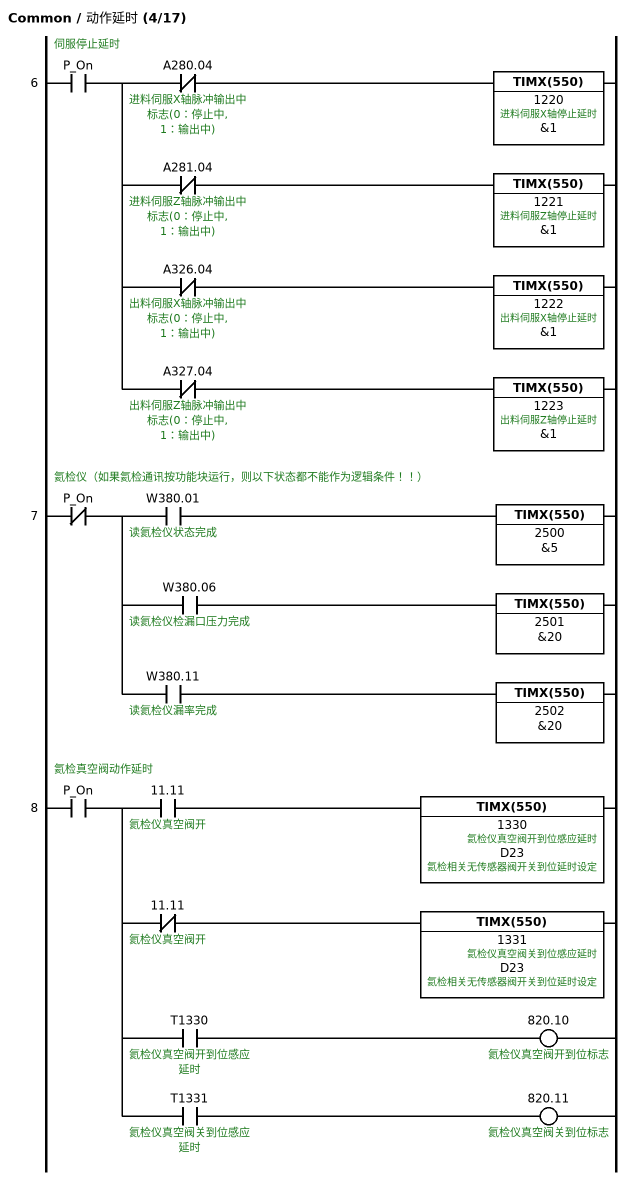
; [picture p480: Common / 动作延时, rungs 6-8]
; rung 6: 伺服停止延时
LD P_On
OUT TR0
ANDNOT A280.04  ; 进料伺服X轴脉冲输出中标志(0：停止中,1：输出中)
TIMX(550) 1220 &1  ; 进料伺服X轴停止延时
LD TR0
ANDNOT A281.04  ; 进料伺服Z轴脉冲输出中标志(0：停止中,1：输出中)
TIMX(550) 1221 &1  ; 进料伺服Z轴停止延时
LD TR0
ANDNOT A326.04  ; 出料伺服X轴脉冲输出中标志(0：停止中,1：输出中)
TIMX(550) 1222 &1  ; 出料伺服X轴停止延时
LD TR0
ANDNOT A327.04  ; 出料伺服Z轴脉冲输出中标志(0：停止中,1：输出中)
TIMX(550) 1223 &1  ; 出料伺服Z轴停止延时
; rung 7: 氦检仪（如果氦检通讯按功能块运行，则以下状态都不能作为逻辑条件！！）
LDNOT P_On
OUT TR0
AND W380.01  ; 读氦检仪状态完成
TIMX(550) 2500 &5
LD TR0
AND W380.06  ; 读氦检仪检漏口压力完成
TIMX(550) 2501 &20
LD TR0
AND W380.11  ; 读氦检仪漏率完成
TIMX(550) 2502 &20
; rung 8: 氦检真空阀动作延时
LD P_On
OUT TR0
AND 11.11  ; 氦检仪真空阀开
TIMX(550) 1330 D23  ; 氦检相关无传感器阀开关到位延时设定, 氦检仪真空阀开到位感应延时
LD TR0
ANDNOT 11.11  ; 氦检仪真空阀开
TIMX(550) 1331 D23  ; 氦检相关无传感器阀开关到位延时设定, 氦检仪真空阀关到位感应延时
LD TR0
AND T1330  ; 氦检仪真空阀开到位感应延时
OUT 820.10  ; 氦检仪真空阀开到位标志
LD TR0
AND T1331  ; 氦检仪真空阀关到位感应延时
OUT 820.11  ; 氦检仪真空阀关到位标志

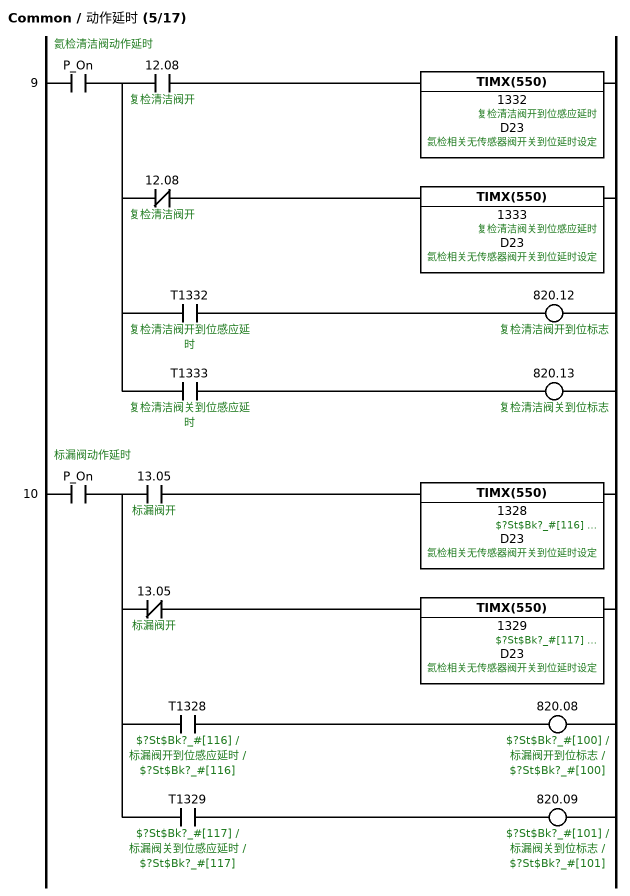
; rung 9: 氦检清洁阀动作延时
LD P_On
OUT TR0
AND 12.08  ; 复检清洁阀开
TIMX(550) 1332 D23  ; 氦检相关无传感器阀开关到位延时设定, 复检清洁阀开到位感应延时
LD TR0
ANDNOT 12.08  ; 复检清洁阀开
TIMX(550) 1333 D23  ; 氦检相关无传感器阀开关到位延时设定, 复检清洁阀关到位感应延时
LD TR0
AND T1332  ; 复检清洁阀开到位感应延时
OUT 820.12  ; 复检清洁阀开到位标志
LD TR0
AND T1333  ; 复检清洁阀关到位感应延时
OUT 820.13  ; 复检清洁阀关到位标志
; rung 10: 标漏阀动作延时
LD P_On
OUT TR0
AND 13.05  ; 标漏阀开
TIMX(550) 1328 D23  ; 氦检相关无传感器阀开关到位延时设定, $?St$Bk?_#[116] / 标漏阀开到位感应延时 / $?St$Bk?_#[116]
LD TR0
ANDNOT 13.05  ; 标漏阀开
TIMX(550) 1329 D23  ; 氦检相关无传感器阀开关到位延时设定, $?St$Bk?_#[117] / 标漏阀关到位感应延时 / $?St$Bk?_#[117]
LD TR0
AND T1328  ; $?St$Bk?_#[116] / 标漏阀开到位感应延时 / $?St$Bk?_#[116]
OUT 820.08  ; $?St$Bk?_#[100] / 标漏阀开到位标志 / $?St$Bk?_#[100]
LD TR0
AND T1329  ; $?St$Bk?_#[117] / 标漏阀关到位感应延时 / $?St$Bk?_#[117]
OUT 820.09  ; $?St$Bk?_#[101] / 标漏阀关到位标志 / $?St$Bk?_#[101]

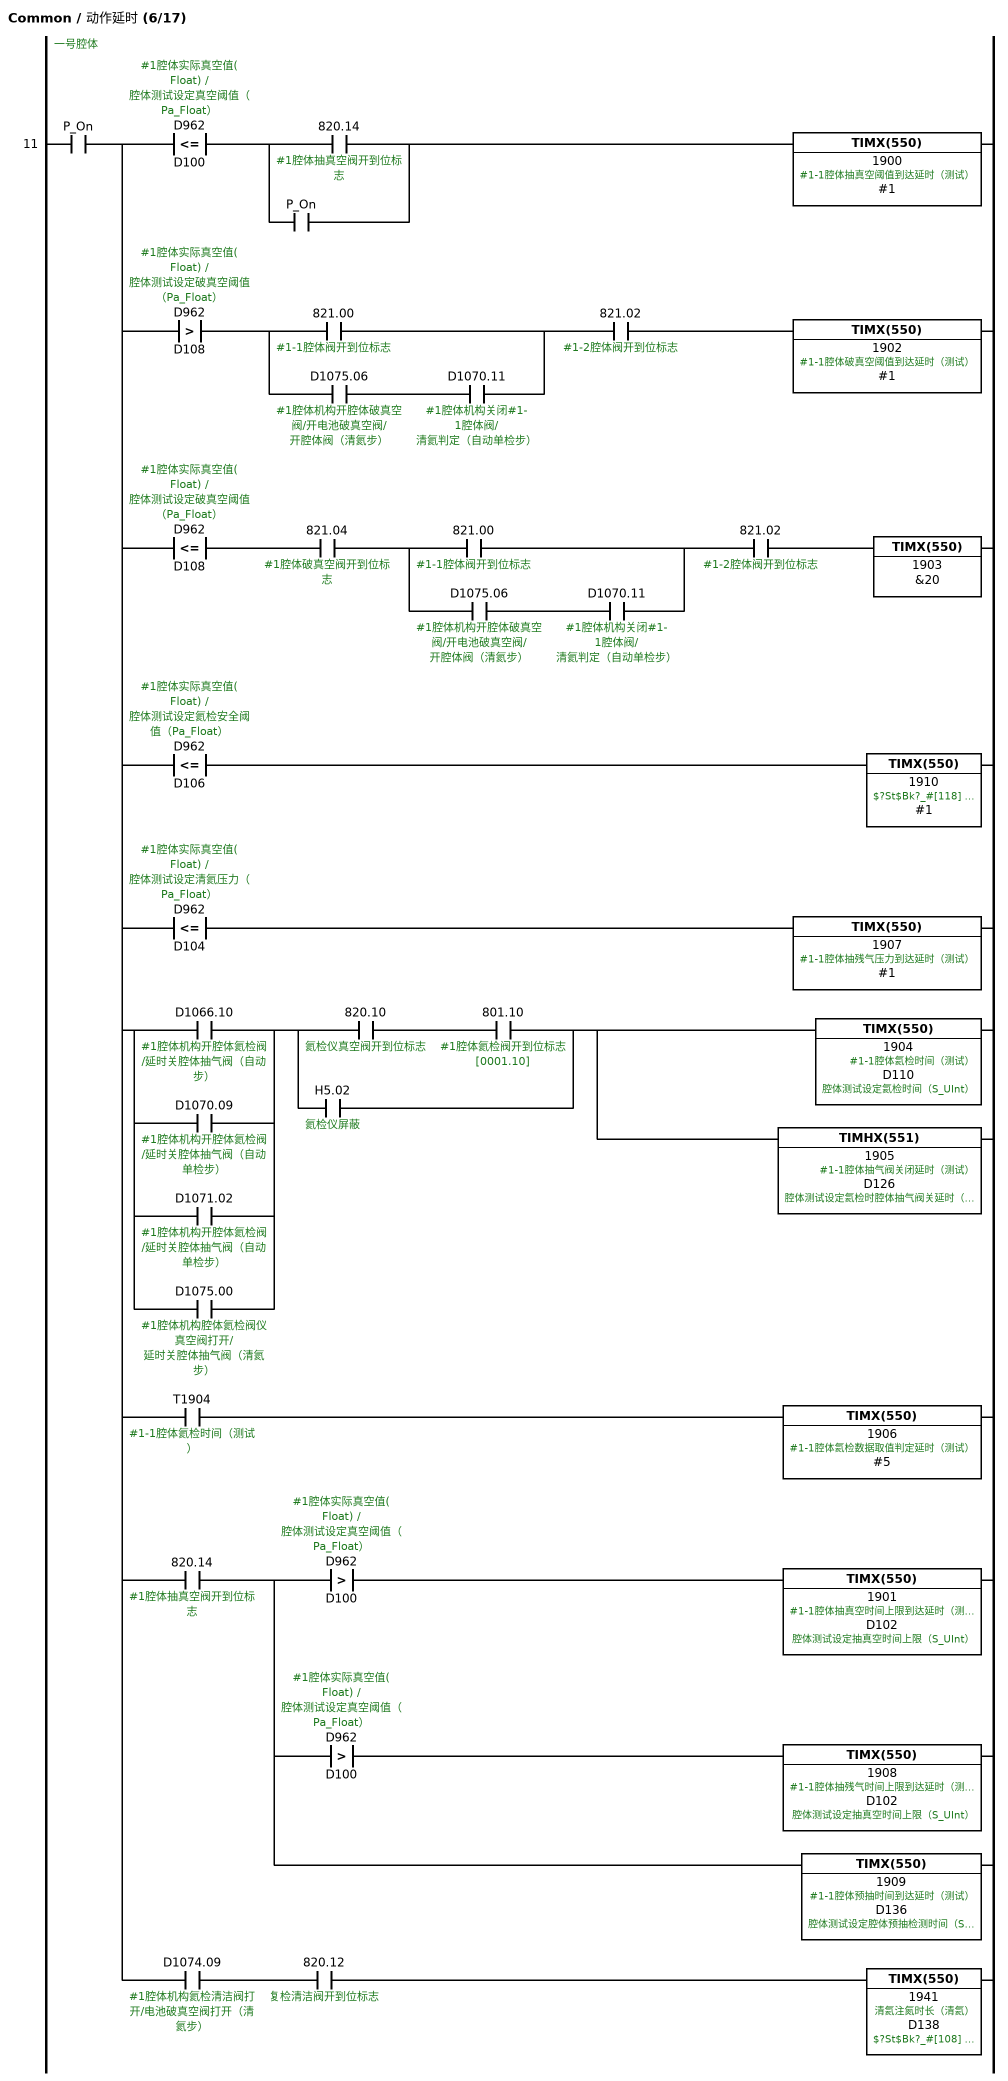
; rung 11: 一号腔体
LD P_On
OUT TR0
AND<=F(332) D962 D100  ; #1腔体实际真空值(Float), 腔体测试设定真空阈值（Pa_Float）
LD 820.14  ; #1腔体抽真空阀开到位标志
OR P_On
ANDLD
TIMX(550) 1900 #1  ; #1-1腔体抽真空阈值到达延时（测试）
LD TR0
AND>F(333) D962 D108  ; #1腔体实际真空值(Float), 腔体测试设定破真空阈值（Pa_Float）
LD 821.00  ; #1-1腔体阀开到位标志
LD D1075.06  ; #1腔体机构开腔体破真空阀/开电池破真空阀/开腔体阀（清氦步）
AND D1070.11  ; #1腔体机构关闭#1-1腔体阀/清氦判定（自动单检步）
ORLD
ANDLD
AND 821.02  ; #1-2腔体阀开到位标志
TIMX(550) 1902 #1  ; #1-1腔体破真空阈值到达延时（测试）
LD TR0
AND<=F(332) D962 D108  ; #1腔体实际真空值(Float), 腔体测试设定破真空阈值（Pa_Float）
AND 821.04  ; #1腔体破真空阀开到位标志
LD 821.00  ; #1-1腔体阀开到位标志
LD D1075.06  ; #1腔体机构开腔体破真空阀/开电池破真空阀/开腔体阀（清氦步）
AND D1070.11  ; #1腔体机构关闭#1-1腔体阀/清氦判定（自动单检步）
ORLD
ANDLD
AND 821.02  ; #1-2腔体阀开到位标志
TIMX(550) 1903 &20
LD TR0
AND<=F(332) D962 D106  ; #1腔体实际真空值(Float), 腔体测试设定氦检安全阈值（Pa_Float）
TIMX(550) 1910 #1  ; $?St$Bk?_#[118] / #1-1腔体真空在可氦检状态（测试） / $?St$Bk?_#[118]
LD TR0
AND<=F(332) D962 D104  ; #1腔体实际真空值(Float), 腔体测试设定清氦压力（Pa_Float）
TIMX(550) 1907 #1  ; #1-1腔体抽残气压力到达延时（测试）
LD TR0
LD D1066.10  ; #1腔体机构开腔体氦检阀/延时关腔体抽气阀（自动步）
OR D1070.09  ; #1腔体机构开腔体氦检阀/延时关腔体抽气阀（自动单检步）
OR D1071.02  ; #1腔体机构开腔体氦检阀/延时关腔体抽气阀（自动单检步）
OR D1075.00  ; #1腔体机构腔体氦检阀仪真空阀打开/延时关腔体抽气阀（清氦步）
ANDLD
LD 820.10  ; 氦检仪真空阀开到位标志
AND 801.10  ; #1腔体氦检阀开到位标志[0001.10]
OR H5.02  ; 氦检仪屏蔽
ANDLD
TIMX(550) 1904 D110  ; 腔体测试设定氦检时间（S_UInt）, #1-1腔体氦检时间（测试）
TIMHX(551) 1905 D126  ; 腔体测试设定氦检时腔体抽气阀关延时（S_UInt）, #1-1腔体抽气阀关闭延时（测试）
LD TR0
AND T1904  ; #1-1腔体氦检时间（测试）
TIMX(550) 1906 #5  ; #1-1腔体氦检数据取值判定延时（测试）
LD TR0
AND 820.14  ; #1腔体抽真空阀开到位标志
OUT TR1
AND>F(333) D962 D100  ; #1腔体实际真空值(Float), 腔体测试设定真空阈值（Pa_Float）
TIMX(550) 1901 D102  ; 腔体测试设定抽真空时间上限（S_UInt）, #1-1腔体抽真空时间上限到达延时（测试）
LD TR1
AND>F(333) D962 D100  ; #1腔体实际真空值(Float), 腔体测试设定真空阈值（Pa_Float）
TIMX(550) 1908 D102  ; 腔体测试设定抽真空时间上限（S_UInt）, #1-1腔体抽残气时间上限到达延时（测试）
LD TR1
TIMX(550) 1909 D136  ; 腔体测试设定腔体预抽检测时间（S_UInt）, #1-1腔体预抽时间到达延时（测试）
LD TR0
AND D1074.09  ; #1腔体机构氦检清洁阀打开/电池破真空阀打开（清氦步）
AND 820.12  ; 复检清洁阀开到位标志
TIMX(550) 1941 D138  ; $?St$Bk?_#[108] / 管路清氦注氮时间（S_UInt） / $?St$Bk?_#[108], 清氦注氮时长（清氦）

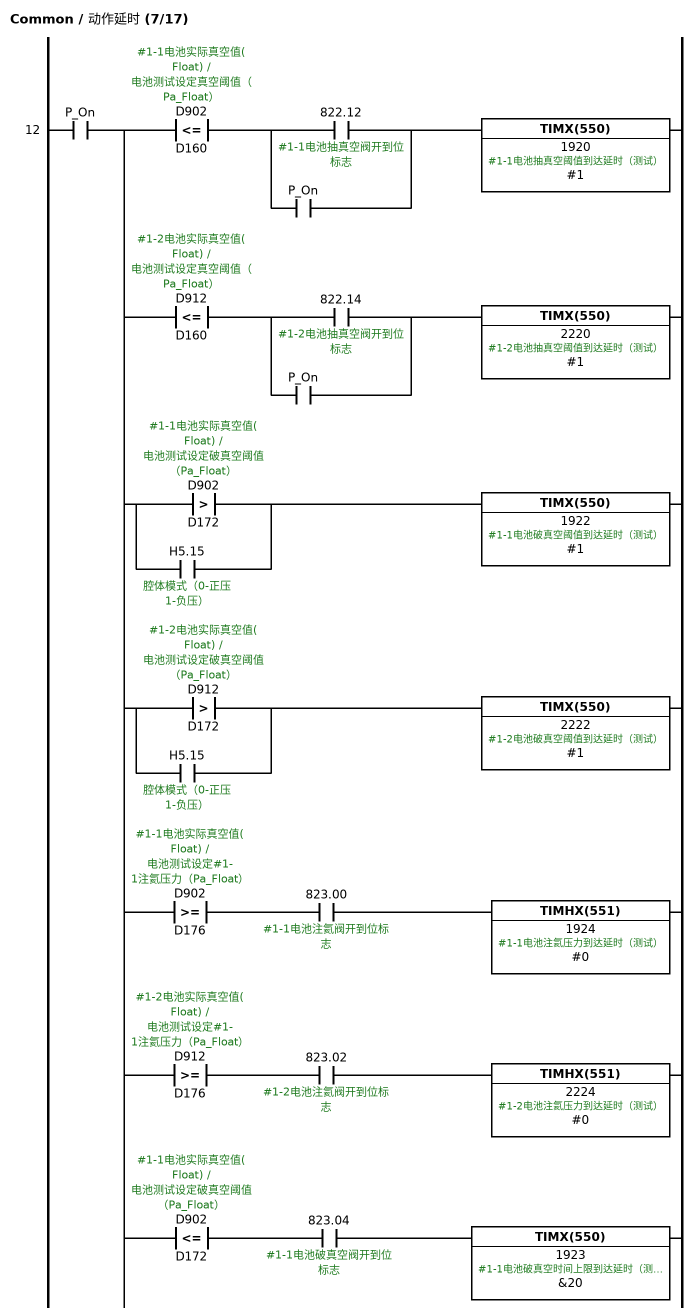

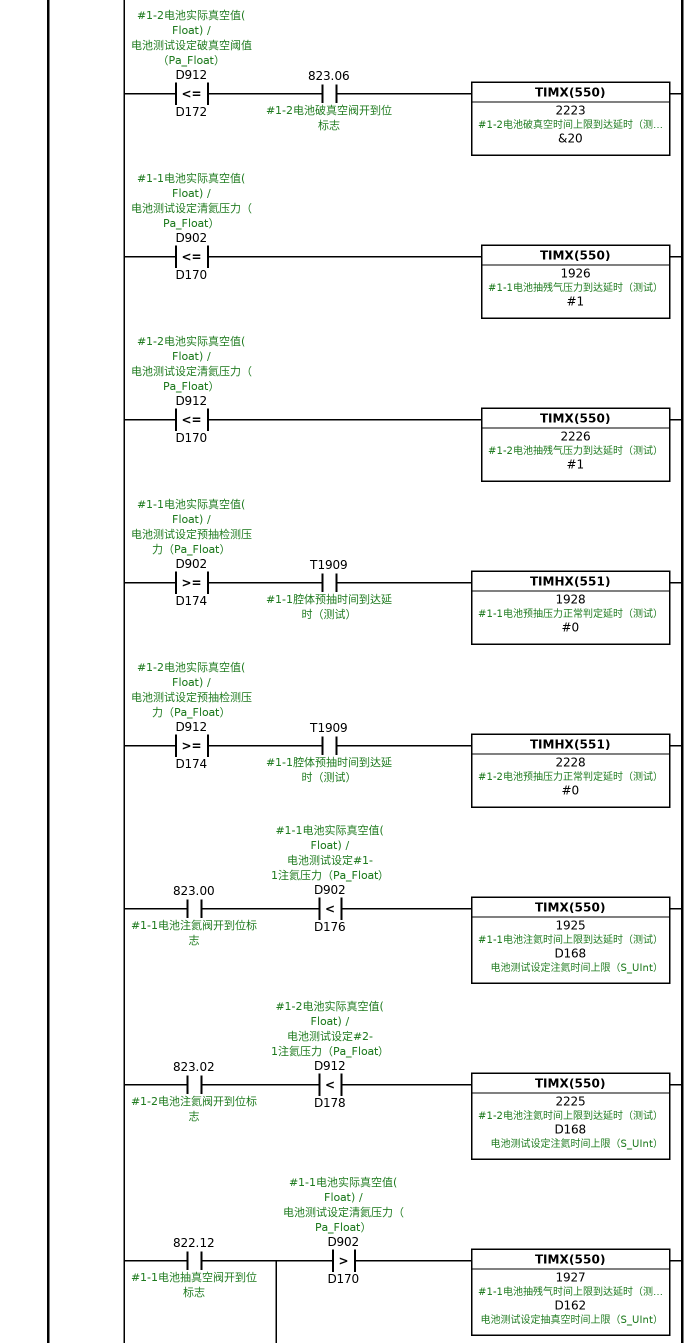

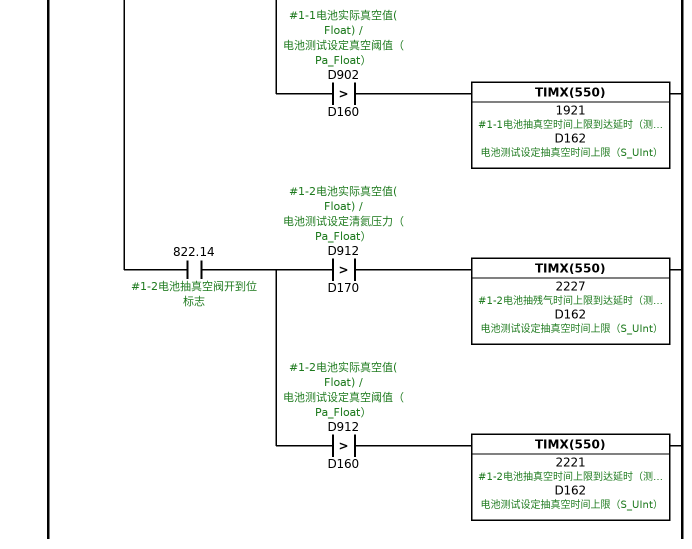
; rung 12
LD P_On
OUT TR0
AND<=F(332) D902 D160  ; #1-1电池实际真空值(Float), 电池测试设定真空阈值（Pa_Float）
LD 822.12  ; #1-1电池抽真空阀开到位标志
OR P_On
ANDLD
TIMX(550) 1920 #1  ; #1-1电池抽真空阈值到达延时（测试）
LD TR0
AND<=F(332) D912 D160  ; #1-2电池实际真空值(Float), 电池测试设定真空阈值（Pa_Float）
LD 822.14  ; #1-2电池抽真空阀开到位标志
OR P_On
ANDLD
TIMX(550) 2220 #1  ; #1-2电池抽真空阈值到达延时（测试）
LD TR0
LD>F(333) D902 D172  ; #1-1电池实际真空值(Float), 电池测试设定破真空阈值（Pa_Float）
OR H5.15  ; 腔体模式（0-正压 1-负压）
ANDLD
TIMX(550) 1922 #1  ; #1-1电池破真空阈值到达延时（测试）
LD TR0
LD>F(333) D912 D172  ; #1-2电池实际真空值(Float), 电池测试设定破真空阈值（Pa_Float）
OR H5.15  ; 腔体模式（0-正压 1-负压）
ANDLD
TIMX(550) 2222 #1  ; #1-2电池破真空阈值到达延时（测试）
LD TR0
AND>=F(334) D902 D176  ; #1-1电池实际真空值(Float), 电池测试设定#1-1注氦压力（Pa_Float）
AND 823.00  ; #1-1电池注氦阀开到位标志
TIMHX(551) 1924 #0  ; #1-1电池注氦压力到达延时（测试）
LD TR0
AND>=F(334) D912 D176  ; #1-2电池实际真空值(Float), 电池测试设定#1-1注氦压力（Pa_Float）
AND 823.02  ; #1-2电池注氦阀开到位标志
TIMHX(551) 2224 #0  ; #1-2电池注氦压力到达延时（测试）
LD TR0
AND<=F(332) D902 D172  ; #1-1电池实际真空值(Float), 电池测试设定破真空阈值（Pa_Float）
AND 823.04  ; #1-1电池破真空阀开到位标志
TIMX(550) 1923 &20  ; #1-1电池破真空时间上限到达延时（测试）
LD TR0
AND<=F(332) D912 D172  ; #1-2电池实际真空值(Float), 电池测试设定破真空阈值（Pa_Float）
AND 823.06  ; #1-2电池破真空阀开到位标志
TIMX(550) 2223 &20  ; #1-2电池破真空时间上限到达延时（测试）
LD TR0
AND<=F(332) D902 D170  ; #1-1电池实际真空值(Float), 电池测试设定清氦压力（Pa_Float）
TIMX(550) 1926 #1  ; #1-1电池抽残气压力到达延时（测试）
LD TR0
AND<=F(332) D912 D170  ; #1-2电池实际真空值(Float), 电池测试设定清氦压力（Pa_Float）
TIMX(550) 2226 #1  ; #1-2电池抽残气压力到达延时（测试）
LD TR0
AND>=F(334) D902 D174  ; #1-1电池实际真空值(Float), 电池测试设定预抽检测压力（Pa_Float）
AND T1909  ; #1-1腔体预抽时间到达延时（测试）
TIMHX(551) 1928 #0  ; #1-1电池预抽压力正常判定延时（测试）
LD TR0
AND>=F(334) D912 D174  ; #1-2电池实际真空值(Float), 电池测试设定预抽检测压力（Pa_Float）
AND T1909  ; #1-1腔体预抽时间到达延时（测试）
TIMHX(551) 2228 #0  ; #1-2电池预抽压力正常判定延时（测试）
LD TR0
AND 823.00  ; #1-1电池注氦阀开到位标志
AND<F(331) D902 D176  ; #1-1电池实际真空值(Float), 电池测试设定#1-1注氦压力（Pa_Float）
TIMX(550) 1925 D168  ; 电池测试设定注氦时间上限（S_UInt）, #1-1电池注氦时间上限到达延时（测试）
LD TR0
AND 823.02  ; #1-2电池注氦阀开到位标志
AND<F(331) D912 D178  ; #1-2电池实际真空值(Float), 电池测试设定#2-1注氦压力（Pa_Float）
TIMX(550) 2225 D168  ; 电池测试设定注氦时间上限（S_UInt）, #1-2电池注氦时间上限到达延时（测试）
LD TR0
AND 822.12  ; #1-1电池抽真空阀开到位标志
OUT TR1
AND>F(333) D902 D170  ; #1-1电池实际真空值(Float), 电池测试设定清氦压力（Pa_Float）
TIMX(550) 1927 D162  ; 电池测试设定抽真空时间上限（S_UInt）, #1-1电池抽残气时间上限到达延时（测试）
LD TR1
AND>F(333) D902 D160  ; #1-1电池实际真空值(Float), 电池测试设定真空阈值（Pa_Float）
TIMX(550) 1921 D162  ; 电池测试设定抽真空时间上限（S_UInt）, #1-1电池抽真空时间上限到达延时（测试）
LD TR0
AND 822.14  ; #1-2电池抽真空阀开到位标志
OUT TR0
AND>F(333) D912 D170  ; #1-2电池实际真空值(Float), 电池测试设定清氦压力（Pa_Float）
TIMX(550) 2227 D162  ; 电池测试设定抽真空时间上限（S_UInt）, #1-2电池抽残气时间上限到达延时（测试）
LD TR0
AND>F(333) D912 D160  ; #1-2电池实际真空值(Float), 电池测试设定真空阈值（Pa_Float）
TIMX(550) 2221 D162  ; 电池测试设定抽真空时间上限（S_UInt）, #1-2电池抽真空时间上限到达延时（测试）

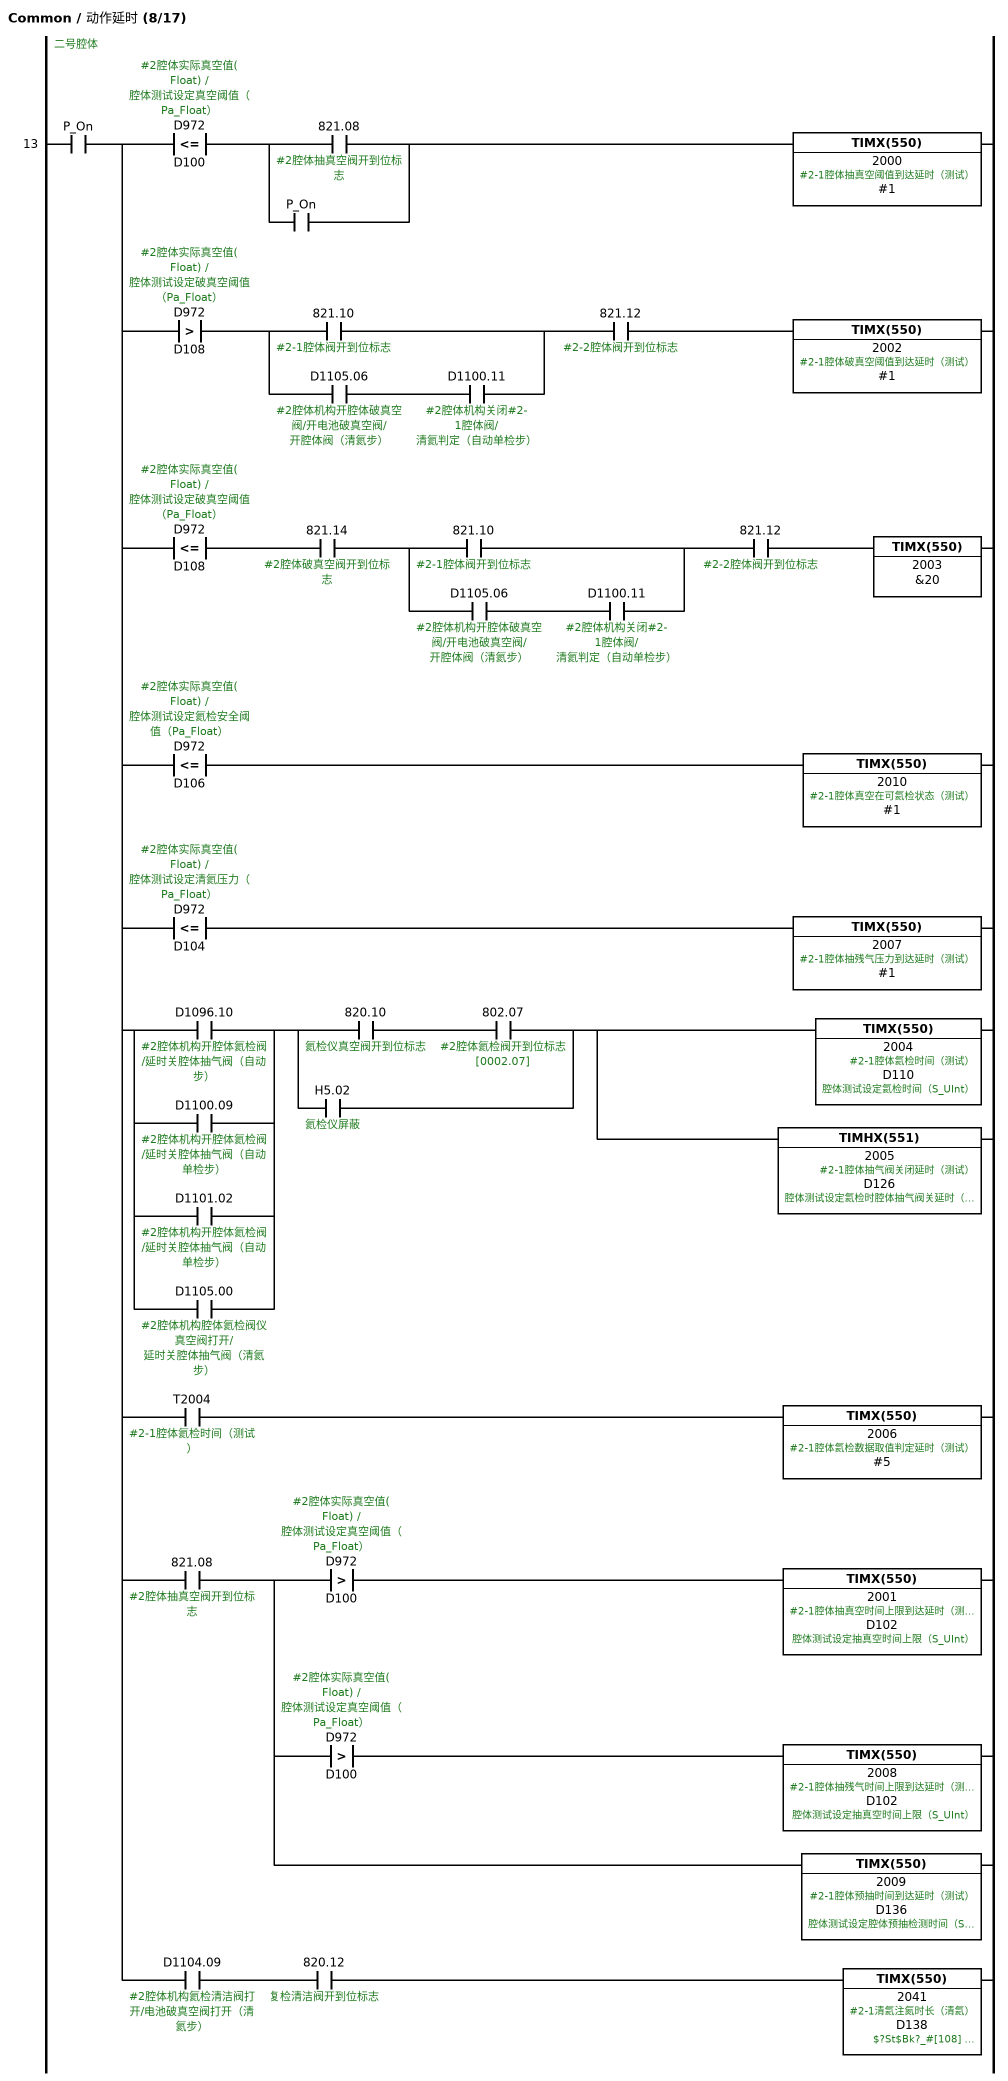
; rung 13: 二号腔体
LD P_On
OUT TR0
AND<=F(332) D972 D100  ; #2腔体实际真空值(Float), 腔体测试设定真空阈值（Pa_Float）
LD 821.08  ; #2腔体抽真空阀开到位标志
OR P_On
ANDLD
TIMX(550) 2000 #1  ; #2-1腔体抽真空阈值到达延时（测试）
LD TR0
AND>F(333) D972 D108  ; #2腔体实际真空值(Float), 腔体测试设定破真空阈值（Pa_Float）
LD 821.10  ; #2-1腔体阀开到位标志
LD D1105.06  ; #2腔体机构开腔体破真空阀/开电池破真空阀/开腔体阀（清氦步）
AND D1100.11  ; #2腔体机构关闭#2-1腔体阀/清氦判定（自动单检步）
ORLD
ANDLD
AND 821.12  ; #2-2腔体阀开到位标志
TIMX(550) 2002 #1  ; #2-1腔体破真空阈值到达延时（测试）
LD TR0
AND<=F(332) D972 D108  ; #2腔体实际真空值(Float), 腔体测试设定破真空阈值（Pa_Float）
AND 821.14  ; #2腔体破真空阀开到位标志
LD 821.10  ; #2-1腔体阀开到位标志
LD D1105.06  ; #2腔体机构开腔体破真空阀/开电池破真空阀/开腔体阀（清氦步）
AND D1100.11  ; #2腔体机构关闭#2-1腔体阀/清氦判定（自动单检步）
ORLD
ANDLD
AND 821.12  ; #2-2腔体阀开到位标志
TIMX(550) 2003 &20
LD TR0
AND<=F(332) D972 D106  ; #2腔体实际真空值(Float), 腔体测试设定氦检安全阈值（Pa_Float）
TIMX(550) 2010 #1  ; #2-1腔体真空在可氦检状态（测试）
LD TR0
AND<=F(332) D972 D104  ; #2腔体实际真空值(Float), 腔体测试设定清氦压力（Pa_Float）
TIMX(550) 2007 #1  ; #2-1腔体抽残气压力到达延时（测试）
LD TR0
LD D1096.10  ; #2腔体机构开腔体氦检阀/延时关腔体抽气阀（自动步）
OR D1100.09  ; #2腔体机构开腔体氦检阀/延时关腔体抽气阀（自动单检步）
OR D1101.02  ; #2腔体机构开腔体氦检阀/延时关腔体抽气阀（自动单检步）
OR D1105.00  ; #2腔体机构腔体氦检阀仪真空阀打开/延时关腔体抽气阀（清氦步）
ANDLD
LD 820.10  ; 氦检仪真空阀开到位标志
AND 802.07  ; #2腔体氦检阀开到位标志[0002.07]
OR H5.02  ; 氦检仪屏蔽
ANDLD
TIMX(550) 2004 D110  ; 腔体测试设定氦检时间（S_UInt）, #2-1腔体氦检时间（测试）
TIMHX(551) 2005 D126  ; 腔体测试设定氦检时腔体抽气阀关延时（S_UInt）, #2-1腔体抽气阀关闭延时（测试）
LD TR0
AND T2004  ; #2-1腔体氦检时间（测试）
TIMX(550) 2006 #5  ; #2-1腔体氦检数据取值判定延时（测试）
LD TR0
AND 821.08  ; #2腔体抽真空阀开到位标志
OUT TR1
AND>F(333) D972 D100  ; #2腔体实际真空值(Float), 腔体测试设定真空阈值（Pa_Float）
TIMX(550) 2001 D102  ; 腔体测试设定抽真空时间上限（S_UInt）, #2-1腔体抽真空时间上限到达延时（测试）
LD TR1
AND>F(333) D972 D100  ; #2腔体实际真空值(Float), 腔体测试设定真空阈值（Pa_Float）
TIMX(550) 2008 D102  ; 腔体测试设定抽真空时间上限（S_UInt）, #2-1腔体抽残气时间上限到达延时（测试）
LD TR1
TIMX(550) 2009 D136  ; 腔体测试设定腔体预抽检测时间（S_UInt）, #2-1腔体预抽时间到达延时（测试）
LD TR0
AND D1104.09  ; #2腔体机构氦检清洁阀打开/电池破真空阀打开（清氦步）
AND 820.12  ; 复检清洁阀开到位标志
TIMX(550) 2041 D138  ; $?St$Bk?_#[108] / 管路清氦注氮时间（S_UInt） / $?St$Bk?_#[108], #2-1清氦注氮时长（清氦）

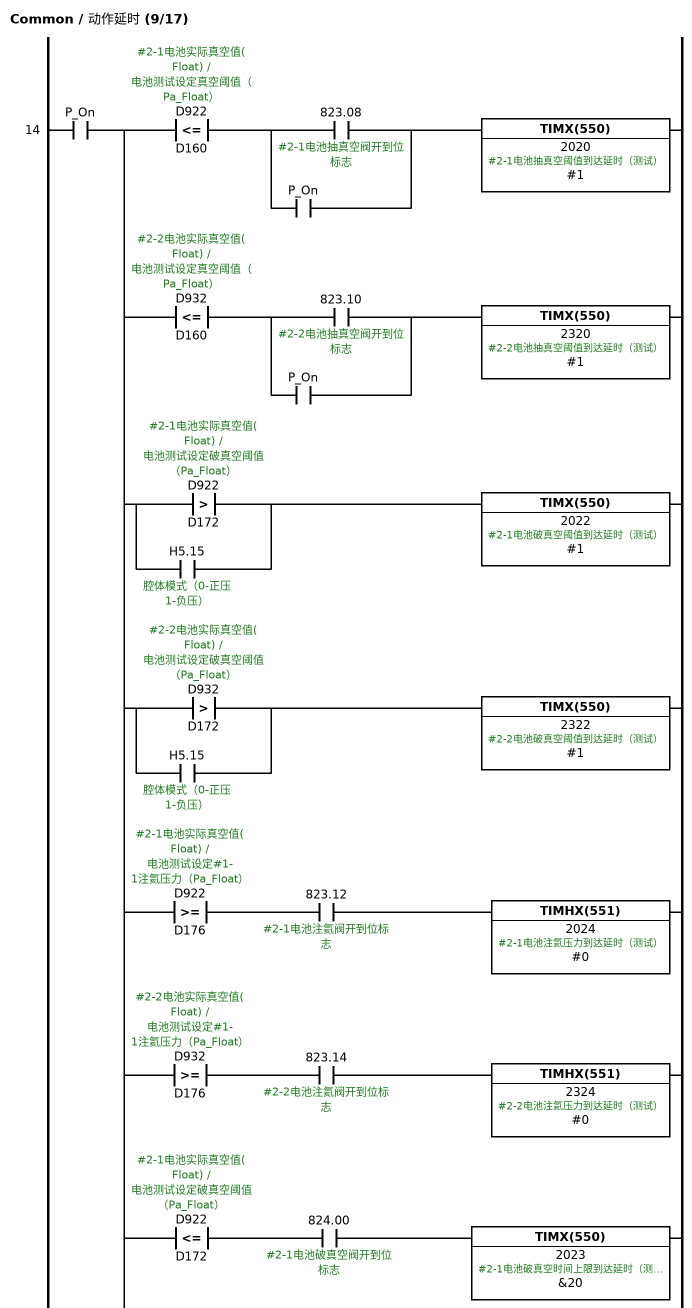

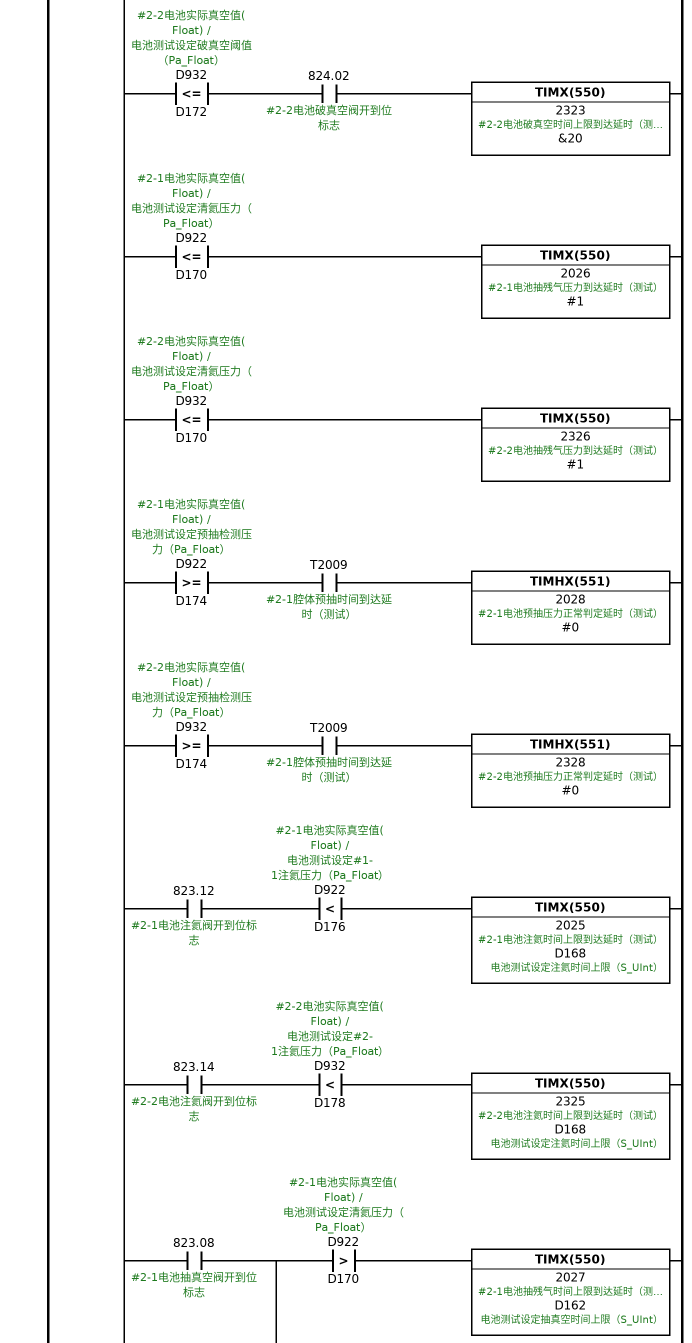

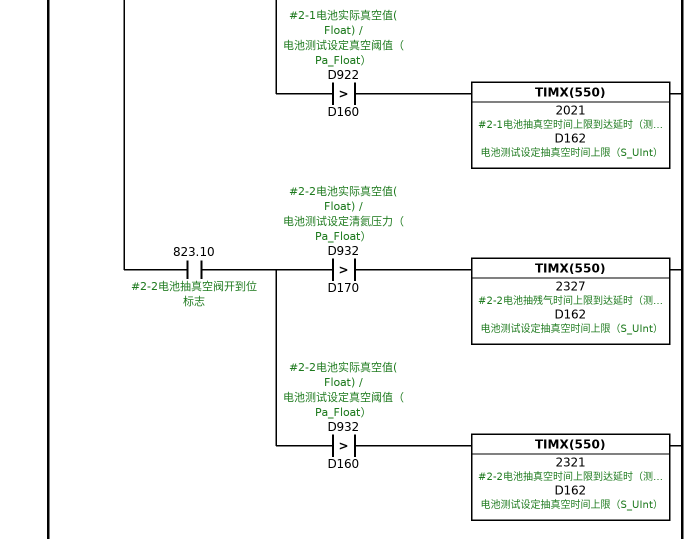
; rung 14
LD P_On
OUT TR0
AND<=F(332) D922 D160  ; #2-1电池实际真空值(Float), 电池测试设定真空阈值（Pa_Float）
LD 823.08  ; #2-1电池抽真空阀开到位标志
OR P_On
ANDLD
TIMX(550) 2020 #1  ; #2-1电池抽真空阈值到达延时（测试）
LD TR0
AND<=F(332) D932 D160  ; #2-2电池实际真空值(Float), 电池测试设定真空阈值（Pa_Float）
LD 823.10  ; #2-2电池抽真空阀开到位标志
OR P_On
ANDLD
TIMX(550) 2320 #1  ; #2-2电池抽真空阈值到达延时（测试）
LD TR0
LD>F(333) D922 D172  ; #2-1电池实际真空值(Float), 电池测试设定破真空阈值（Pa_Float）
OR H5.15  ; 腔体模式（0-正压 1-负压）
ANDLD
TIMX(550) 2022 #1  ; #2-1电池破真空阈值到达延时（测试）
LD TR0
LD>F(333) D932 D172  ; #2-2电池实际真空值(Float), 电池测试设定破真空阈值（Pa_Float）
OR H5.15  ; 腔体模式（0-正压 1-负压）
ANDLD
TIMX(550) 2322 #1  ; #2-2电池破真空阈值到达延时（测试）
LD TR0
AND>=F(334) D922 D176  ; #2-1电池实际真空值(Float), 电池测试设定#1-1注氦压力（Pa_Float）
AND 823.12  ; #2-1电池注氦阀开到位标志
TIMHX(551) 2024 #0  ; #2-1电池注氦压力到达延时（测试）
LD TR0
AND>=F(334) D932 D176  ; #2-2电池实际真空值(Float), 电池测试设定#1-1注氦压力（Pa_Float）
AND 823.14  ; #2-2电池注氦阀开到位标志
TIMHX(551) 2324 #0  ; #2-2电池注氦压力到达延时（测试）
LD TR0
AND<=F(332) D922 D172  ; #2-1电池实际真空值(Float), 电池测试设定破真空阈值（Pa_Float）
AND 824.00  ; #2-1电池破真空阀开到位标志
TIMX(550) 2023 &20  ; #2-1电池破真空时间上限到达延时（测试）
LD TR0
AND<=F(332) D932 D172  ; #2-2电池实际真空值(Float), 电池测试设定破真空阈值（Pa_Float）
AND 824.02  ; #2-2电池破真空阀开到位标志
TIMX(550) 2323 &20  ; #2-2电池破真空时间上限到达延时（测试）
LD TR0
AND<=F(332) D922 D170  ; #2-1电池实际真空值(Float), 电池测试设定清氦压力（Pa_Float）
TIMX(550) 2026 #1  ; #2-1电池抽残气压力到达延时（测试）
LD TR0
AND<=F(332) D932 D170  ; #2-2电池实际真空值(Float), 电池测试设定清氦压力（Pa_Float）
TIMX(550) 2326 #1  ; #2-2电池抽残气压力到达延时（测试）
LD TR0
AND>=F(334) D922 D174  ; #2-1电池实际真空值(Float), 电池测试设定预抽检测压力（Pa_Float）
AND T2009  ; #2-1腔体预抽时间到达延时（测试）
TIMHX(551) 2028 #0  ; #2-1电池预抽压力正常判定延时（测试）
LD TR0
AND>=F(334) D932 D174  ; #2-2电池实际真空值(Float), 电池测试设定预抽检测压力（Pa_Float）
AND T2009  ; #2-1腔体预抽时间到达延时（测试）
TIMHX(551) 2328 #0  ; #2-2电池预抽压力正常判定延时（测试）
LD TR0
AND 823.12  ; #2-1电池注氦阀开到位标志
AND<F(331) D922 D176  ; #2-1电池实际真空值(Float), 电池测试设定#1-1注氦压力（Pa_Float）
TIMX(550) 2025 D168  ; 电池测试设定注氦时间上限（S_UInt）, #2-1电池注氦时间上限到达延时（测试）
LD TR0
AND 823.14  ; #2-2电池注氦阀开到位标志
AND<F(331) D932 D178  ; #2-2电池实际真空值(Float), 电池测试设定#2-1注氦压力（Pa_Float）
TIMX(550) 2325 D168  ; 电池测试设定注氦时间上限（S_UInt）, #2-2电池注氦时间上限到达延时（测试）
LD TR0
AND 823.08  ; #2-1电池抽真空阀开到位标志
OUT TR1
AND>F(333) D922 D170  ; #2-1电池实际真空值(Float), 电池测试设定清氦压力（Pa_Float）
TIMX(550) 2027 D162  ; 电池测试设定抽真空时间上限（S_UInt）, #2-1电池抽残气时间上限到达延时（测试）
LD TR1
AND>F(333) D922 D160  ; #2-1电池实际真空值(Float), 电池测试设定真空阈值（Pa_Float）
TIMX(550) 2021 D162  ; 电池测试设定抽真空时间上限（S_UInt）, #2-1电池抽真空时间上限到达延时（测试）
LD TR0
AND 823.10  ; #2-2电池抽真空阀开到位标志
OUT TR0
AND>F(333) D932 D170  ; #2-2电池实际真空值(Float), 电池测试设定清氦压力（Pa_Float）
TIMX(550) 2327 D162  ; 电池测试设定抽真空时间上限（S_UInt）, #2-2电池抽残气时间上限到达延时（测试）
LD TR0
AND>F(333) D932 D160  ; #2-2电池实际真空值(Float), 电池测试设定真空阈值（Pa_Float）
TIMX(550) 2321 D162  ; 电池测试设定抽真空时间上限（S_UInt）, #2-2电池抽真空时间上限到达延时（测试）

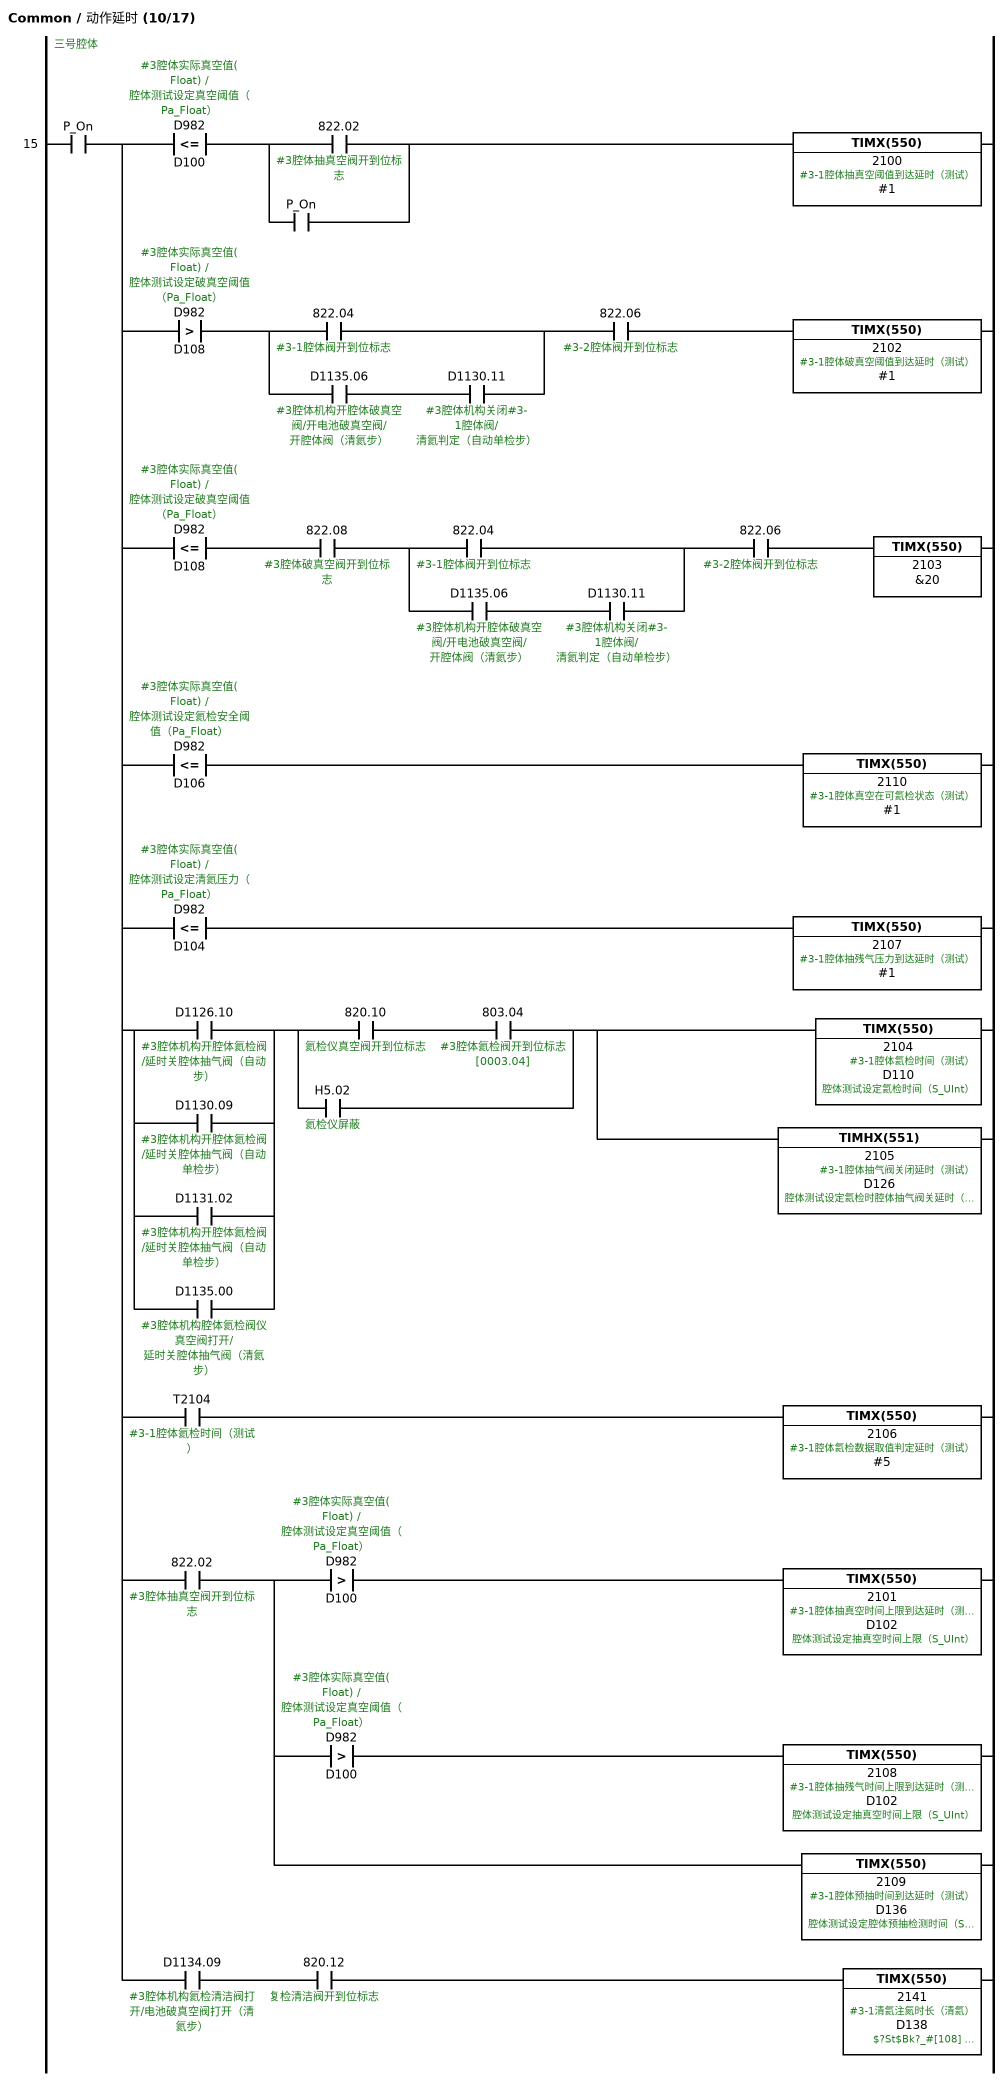
; rung 15: 三号腔体
LD P_On
OUT TR0
AND<=F(332) D982 D100  ; #3腔体实际真空值(Float), 腔体测试设定真空阈值（Pa_Float）
LD 822.02  ; #3腔体抽真空阀开到位标志
OR P_On
ANDLD
TIMX(550) 2100 #1  ; #3-1腔体抽真空阈值到达延时（测试）
LD TR0
AND>F(333) D982 D108  ; #3腔体实际真空值(Float), 腔体测试设定破真空阈值（Pa_Float）
LD 822.04  ; #3-1腔体阀开到位标志
LD D1135.06  ; #3腔体机构开腔体破真空阀/开电池破真空阀/开腔体阀（清氦步）
AND D1130.11  ; #3腔体机构关闭#3-1腔体阀/清氦判定（自动单检步）
ORLD
ANDLD
AND 822.06  ; #3-2腔体阀开到位标志
TIMX(550) 2102 #1  ; #3-1腔体破真空阈值到达延时（测试）
LD TR0
AND<=F(332) D982 D108  ; #3腔体实际真空值(Float), 腔体测试设定破真空阈值（Pa_Float）
AND 822.08  ; #3腔体破真空阀开到位标志
LD 822.04  ; #3-1腔体阀开到位标志
LD D1135.06  ; #3腔体机构开腔体破真空阀/开电池破真空阀/开腔体阀（清氦步）
AND D1130.11  ; #3腔体机构关闭#3-1腔体阀/清氦判定（自动单检步）
ORLD
ANDLD
AND 822.06  ; #3-2腔体阀开到位标志
TIMX(550) 2103 &20
LD TR0
AND<=F(332) D982 D106  ; #3腔体实际真空值(Float), 腔体测试设定氦检安全阈值（Pa_Float）
TIMX(550) 2110 #1  ; #3-1腔体真空在可氦检状态（测试）
LD TR0
AND<=F(332) D982 D104  ; #3腔体实际真空值(Float), 腔体测试设定清氦压力（Pa_Float）
TIMX(550) 2107 #1  ; #3-1腔体抽残气压力到达延时（测试）
LD TR0
LD D1126.10  ; #3腔体机构开腔体氦检阀/延时关腔体抽气阀（自动步）
OR D1130.09  ; #3腔体机构开腔体氦检阀/延时关腔体抽气阀（自动单检步）
OR D1131.02  ; #3腔体机构开腔体氦检阀/延时关腔体抽气阀（自动单检步）
OR D1135.00  ; #3腔体机构腔体氦检阀仪真空阀打开/延时关腔体抽气阀（清氦步）
ANDLD
LD 820.10  ; 氦检仪真空阀开到位标志
AND 803.04  ; #3腔体氦检阀开到位标志[0003.04]
OR H5.02  ; 氦检仪屏蔽
ANDLD
TIMX(550) 2104 D110  ; 腔体测试设定氦检时间（S_UInt）, #3-1腔体氦检时间（测试）
TIMHX(551) 2105 D126  ; 腔体测试设定氦检时腔体抽气阀关延时（S_UInt）, #3-1腔体抽气阀关闭延时（测试）
LD TR0
AND T2104  ; #3-1腔体氦检时间（测试）
TIMX(550) 2106 #5  ; #3-1腔体氦检数据取值判定延时（测试）
LD TR0
AND 822.02  ; #3腔体抽真空阀开到位标志
OUT TR1
AND>F(333) D982 D100  ; #3腔体实际真空值(Float), 腔体测试设定真空阈值（Pa_Float）
TIMX(550) 2101 D102  ; 腔体测试设定抽真空时间上限（S_UInt）, #3-1腔体抽真空时间上限到达延时（测试）
LD TR1
AND>F(333) D982 D100  ; #3腔体实际真空值(Float), 腔体测试设定真空阈值（Pa_Float）
TIMX(550) 2108 D102  ; 腔体测试设定抽真空时间上限（S_UInt）, #3-1腔体抽残气时间上限到达延时（测试）
LD TR1
TIMX(550) 2109 D136  ; 腔体测试设定腔体预抽检测时间（S_UInt）, #3-1腔体预抽时间到达延时（测试）
LD TR0
AND D1134.09  ; #3腔体机构氦检清洁阀打开/电池破真空阀打开（清氦步）
AND 820.12  ; 复检清洁阀开到位标志
TIMX(550) 2141 D138  ; $?St$Bk?_#[108] / 管路清氦注氮时间（S_UInt） / $?St$Bk?_#[108], #3-1清氦注氮时长（清氦）

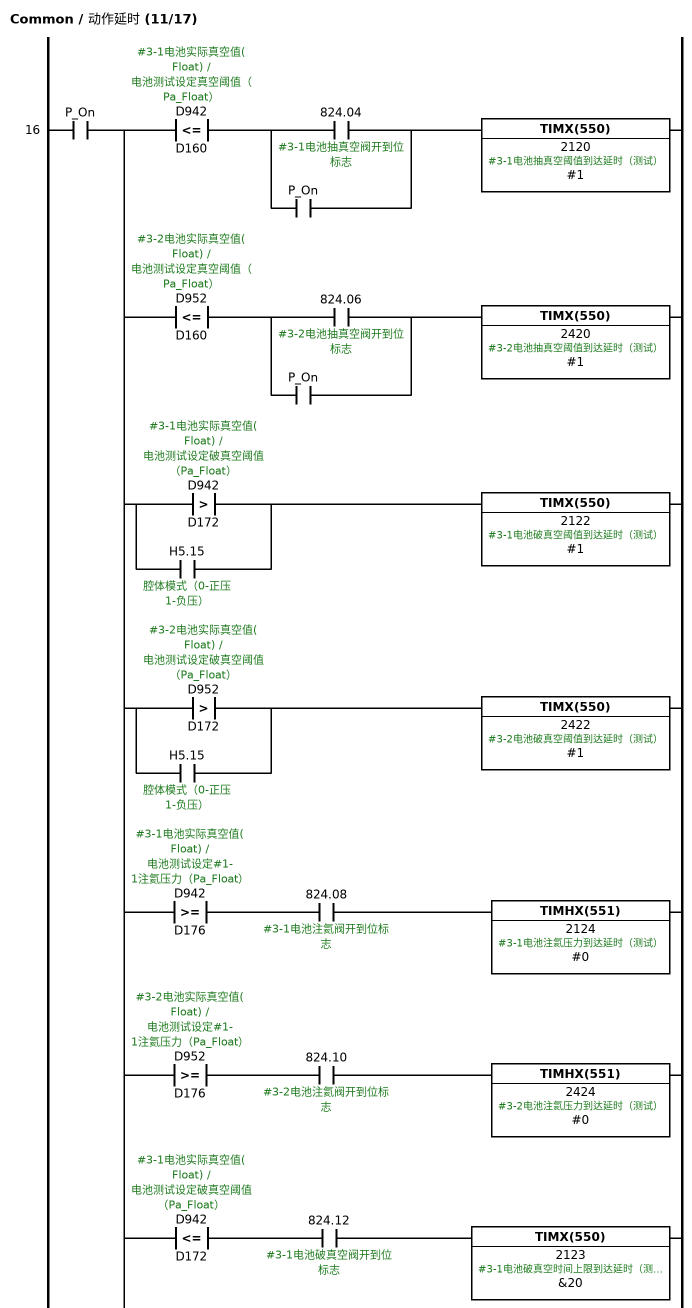

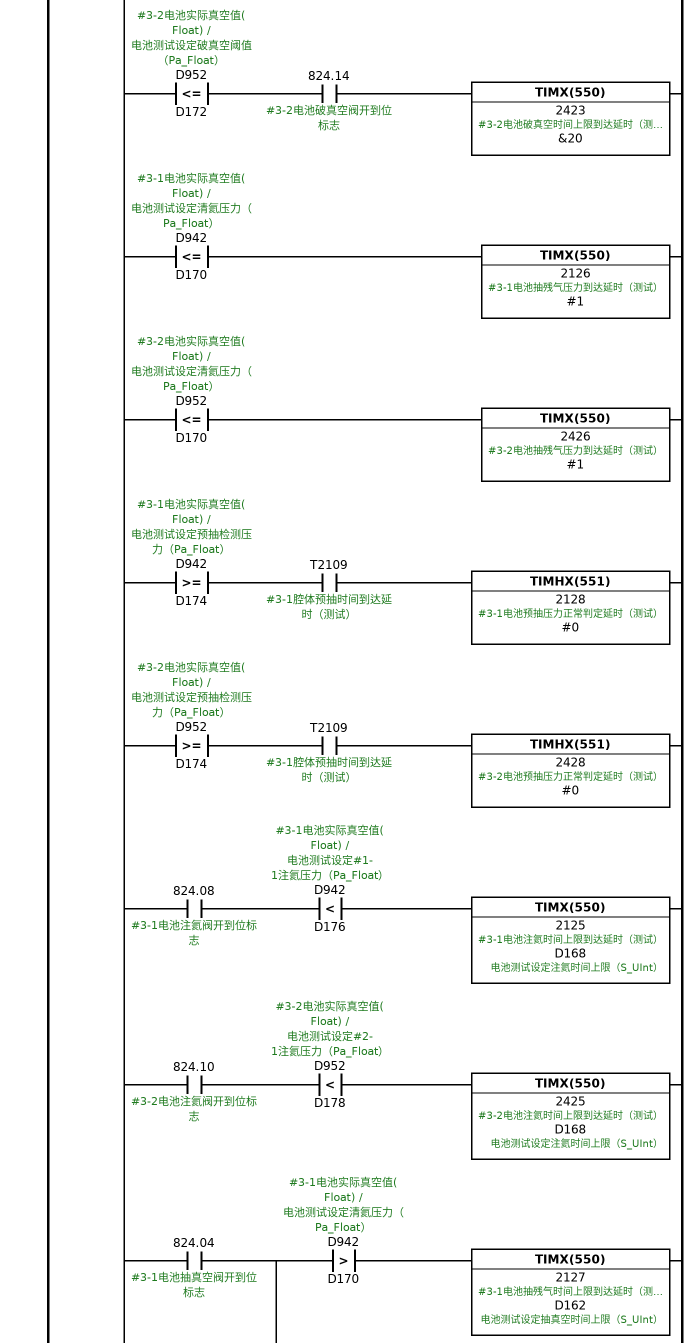

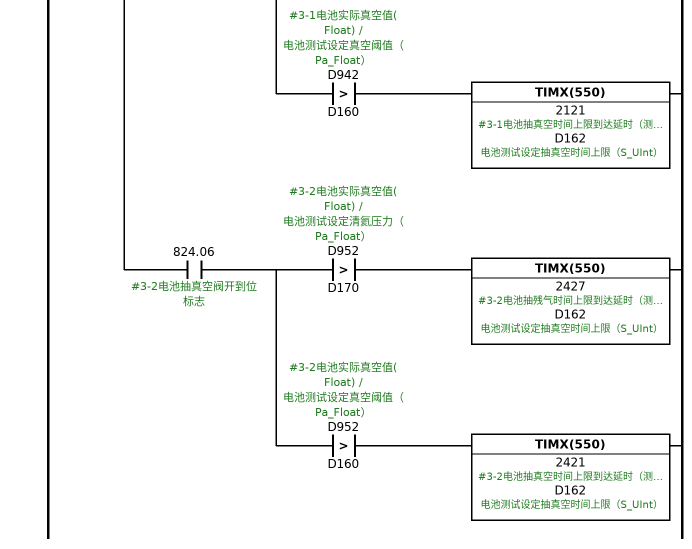
; rung 16
LD P_On
OUT TR0
AND<=F(332) D942 D160  ; #3-1电池实际真空值(Float), 电池测试设定真空阈值（Pa_Float）
LD 824.04  ; #3-1电池抽真空阀开到位标志
OR P_On
ANDLD
TIMX(550) 2120 #1  ; #3-1电池抽真空阈值到达延时（测试）
LD TR0
AND<=F(332) D952 D160  ; #3-2电池实际真空值(Float), 电池测试设定真空阈值（Pa_Float）
LD 824.06  ; #3-2电池抽真空阀开到位标志
OR P_On
ANDLD
TIMX(550) 2420 #1  ; #3-2电池抽真空阈值到达延时（测试）
LD TR0
LD>F(333) D942 D172  ; #3-1电池实际真空值(Float), 电池测试设定破真空阈值（Pa_Float）
OR H5.15  ; 腔体模式（0-正压 1-负压）
ANDLD
TIMX(550) 2122 #1  ; #3-1电池破真空阈值到达延时（测试）
LD TR0
LD>F(333) D952 D172  ; #3-2电池实际真空值(Float), 电池测试设定破真空阈值（Pa_Float）
OR H5.15  ; 腔体模式（0-正压 1-负压）
ANDLD
TIMX(550) 2422 #1  ; #3-2电池破真空阈值到达延时（测试）
LD TR0
AND>=F(334) D942 D176  ; #3-1电池实际真空值(Float), 电池测试设定#1-1注氦压力（Pa_Float）
AND 824.08  ; #3-1电池注氦阀开到位标志
TIMHX(551) 2124 #0  ; #3-1电池注氦压力到达延时（测试）
LD TR0
AND>=F(334) D952 D176  ; #3-2电池实际真空值(Float), 电池测试设定#1-1注氦压力（Pa_Float）
AND 824.10  ; #3-2电池注氦阀开到位标志
TIMHX(551) 2424 #0  ; #3-2电池注氦压力到达延时（测试）
LD TR0
AND<=F(332) D942 D172  ; #3-1电池实际真空值(Float), 电池测试设定破真空阈值（Pa_Float）
AND 824.12  ; #3-1电池破真空阀开到位标志
TIMX(550) 2123 &20  ; #3-1电池破真空时间上限到达延时（测试）
LD TR0
AND<=F(332) D952 D172  ; #3-2电池实际真空值(Float), 电池测试设定破真空阈值（Pa_Float）
AND 824.14  ; #3-2电池破真空阀开到位标志
TIMX(550) 2423 &20  ; #3-2电池破真空时间上限到达延时（测试）
LD TR0
AND<=F(332) D942 D170  ; #3-1电池实际真空值(Float), 电池测试设定清氦压力（Pa_Float）
TIMX(550) 2126 #1  ; #3-1电池抽残气压力到达延时（测试）
LD TR0
AND<=F(332) D952 D170  ; #3-2电池实际真空值(Float), 电池测试设定清氦压力（Pa_Float）
TIMX(550) 2426 #1  ; #3-2电池抽残气压力到达延时（测试）
LD TR0
AND>=F(334) D942 D174  ; #3-1电池实际真空值(Float), 电池测试设定预抽检测压力（Pa_Float）
AND T2109  ; #3-1腔体预抽时间到达延时（测试）
TIMHX(551) 2128 #0  ; #3-1电池预抽压力正常判定延时（测试）
LD TR0
AND>=F(334) D952 D174  ; #3-2电池实际真空值(Float), 电池测试设定预抽检测压力（Pa_Float）
AND T2109  ; #3-1腔体预抽时间到达延时（测试）
TIMHX(551) 2428 #0  ; #3-2电池预抽压力正常判定延时（测试）
LD TR0
AND 824.08  ; #3-1电池注氦阀开到位标志
AND<F(331) D942 D176  ; #3-1电池实际真空值(Float), 电池测试设定#1-1注氦压力（Pa_Float）
TIMX(550) 2125 D168  ; 电池测试设定注氦时间上限（S_UInt）, #3-1电池注氦时间上限到达延时（测试）
LD TR0
AND 824.10  ; #3-2电池注氦阀开到位标志
AND<F(331) D952 D178  ; #3-2电池实际真空值(Float), 电池测试设定#2-1注氦压力（Pa_Float）
TIMX(550) 2425 D168  ; 电池测试设定注氦时间上限（S_UInt）, #3-2电池注氦时间上限到达延时（测试）
LD TR0
AND 824.04  ; #3-1电池抽真空阀开到位标志
OUT TR1
AND>F(333) D942 D170  ; #3-1电池实际真空值(Float), 电池测试设定清氦压力（Pa_Float）
TIMX(550) 2127 D162  ; 电池测试设定抽真空时间上限（S_UInt）, #3-1电池抽残气时间上限到达延时（测试）
LD TR1
AND>F(333) D942 D160  ; #3-1电池实际真空值(Float), 电池测试设定真空阈值（Pa_Float）
TIMX(550) 2121 D162  ; 电池测试设定抽真空时间上限（S_UInt）, #3-1电池抽真空时间上限到达延时（测试）
LD TR0
AND 824.06  ; #3-2电池抽真空阀开到位标志
OUT TR0
AND>F(333) D952 D170  ; #3-2电池实际真空值(Float), 电池测试设定清氦压力（Pa_Float）
TIMX(550) 2427 D162  ; 电池测试设定抽真空时间上限（S_UInt）, #3-2电池抽残气时间上限到达延时（测试）
LD TR0
AND>F(333) D952 D160  ; #3-2电池实际真空值(Float), 电池测试设定真空阈值（Pa_Float）
TIMX(550) 2421 D162  ; 电池测试设定抽真空时间上限（S_UInt）, #3-2电池抽真空时间上限到达延时（测试）

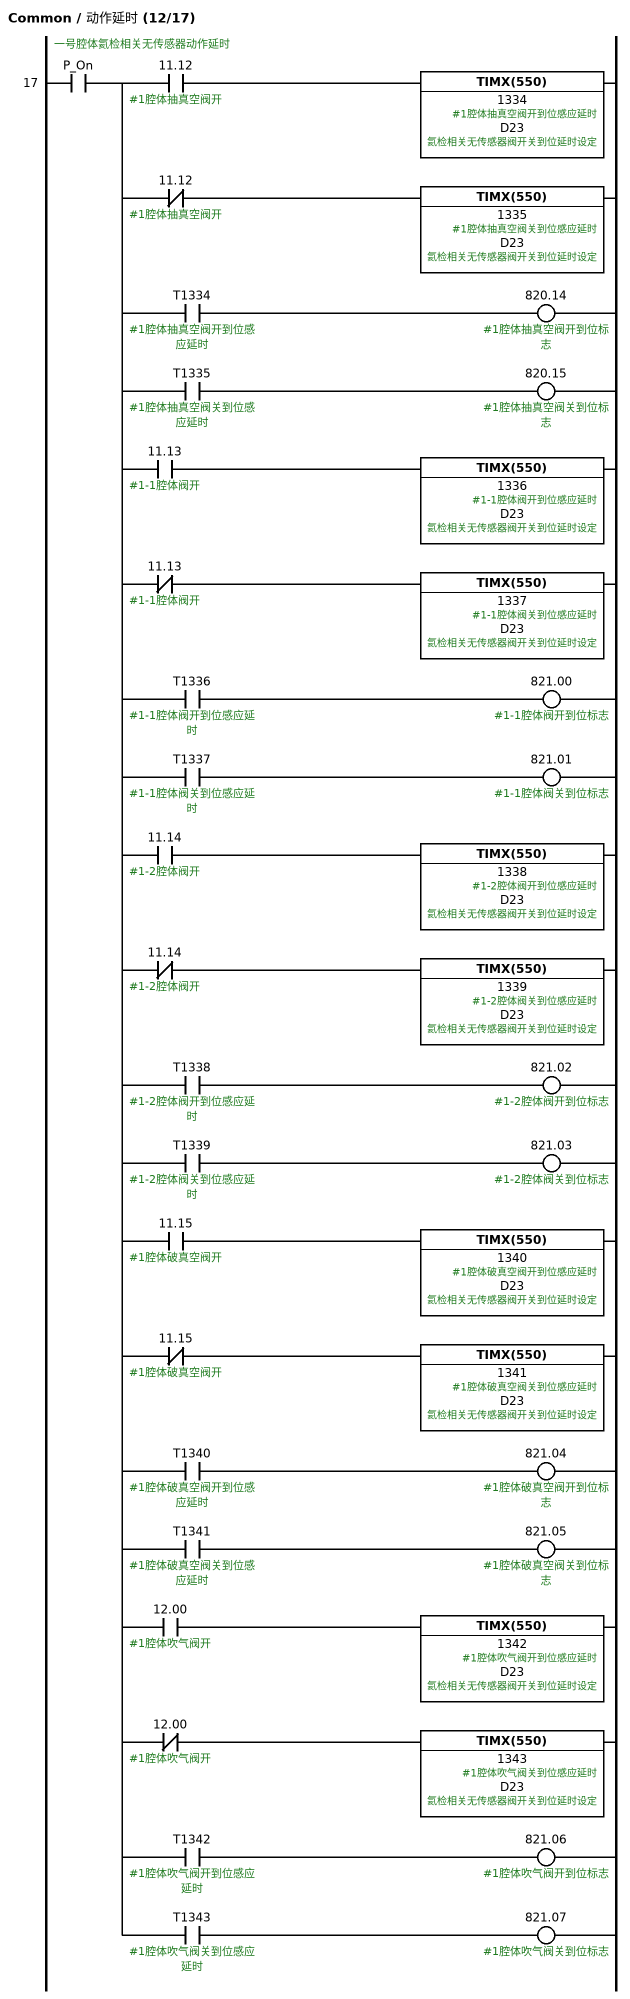
; rung 17: 一号腔体氦检相关无传感器动作延时
LD P_On
OUT TR0
AND 11.12  ; #1腔体抽真空阀开
TIMX(550) 1334 D23  ; 氦检相关无传感器阀开关到位延时设定, #1腔体抽真空阀开到位感应延时
LD TR0
ANDNOT 11.12  ; #1腔体抽真空阀开
TIMX(550) 1335 D23  ; 氦检相关无传感器阀开关到位延时设定, #1腔体抽真空阀关到位感应延时
LD TR0
AND T1334  ; #1腔体抽真空阀开到位感应延时
OUT 820.14  ; #1腔体抽真空阀开到位标志
LD TR0
AND T1335  ; #1腔体抽真空阀关到位感应延时
OUT 820.15  ; #1腔体抽真空阀关到位标志
LD TR0
AND 11.13  ; #1-1腔体阀开
TIMX(550) 1336 D23  ; 氦检相关无传感器阀开关到位延时设定, #1-1腔体阀开到位感应延时
LD TR0
ANDNOT 11.13  ; #1-1腔体阀开
TIMX(550) 1337 D23  ; 氦检相关无传感器阀开关到位延时设定, #1-1腔体阀关到位感应延时
LD TR0
AND T1336  ; #1-1腔体阀开到位感应延时
OUT 821.00  ; #1-1腔体阀开到位标志
LD TR0
AND T1337  ; #1-1腔体阀关到位感应延时
OUT 821.01  ; #1-1腔体阀关到位标志
LD TR0
AND 11.14  ; #1-2腔体阀开
TIMX(550) 1338 D23  ; 氦检相关无传感器阀开关到位延时设定, #1-2腔体阀开到位感应延时
LD TR0
ANDNOT 11.14  ; #1-2腔体阀开
TIMX(550) 1339 D23  ; 氦检相关无传感器阀开关到位延时设定, #1-2腔体阀关到位感应延时
LD TR0
AND T1338  ; #1-2腔体阀开到位感应延时
OUT 821.02  ; #1-2腔体阀开到位标志
LD TR0
AND T1339  ; #1-2腔体阀关到位感应延时
OUT 821.03  ; #1-2腔体阀关到位标志
LD TR0
AND 11.15  ; #1腔体破真空阀开
TIMX(550) 1340 D23  ; 氦检相关无传感器阀开关到位延时设定, #1腔体破真空阀开到位感应延时
LD TR0
ANDNOT 11.15  ; #1腔体破真空阀开
TIMX(550) 1341 D23  ; 氦检相关无传感器阀开关到位延时设定, #1腔体破真空阀关到位感应延时
LD TR0
AND T1340  ; #1腔体破真空阀开到位感应延时
OUT 821.04  ; #1腔体破真空阀开到位标志
LD TR0
AND T1341  ; #1腔体破真空阀关到位感应延时
OUT 821.05  ; #1腔体破真空阀关到位标志
LD TR0
AND 12.00  ; #1腔体吹气阀开
TIMX(550) 1342 D23  ; 氦检相关无传感器阀开关到位延时设定, #1腔体吹气阀开到位感应延时
LD TR0
ANDNOT 12.00  ; #1腔体吹气阀开
TIMX(550) 1343 D23  ; 氦检相关无传感器阀开关到位延时设定, #1腔体吹气阀关到位感应延时
LD TR0
AND T1342  ; #1腔体吹气阀开到位感应延时
OUT 821.06  ; #1腔体吹气阀开到位标志
LD TR0
AND T1343  ; #1腔体吹气阀关到位感应延时
OUT 821.07  ; #1腔体吹气阀关到位标志

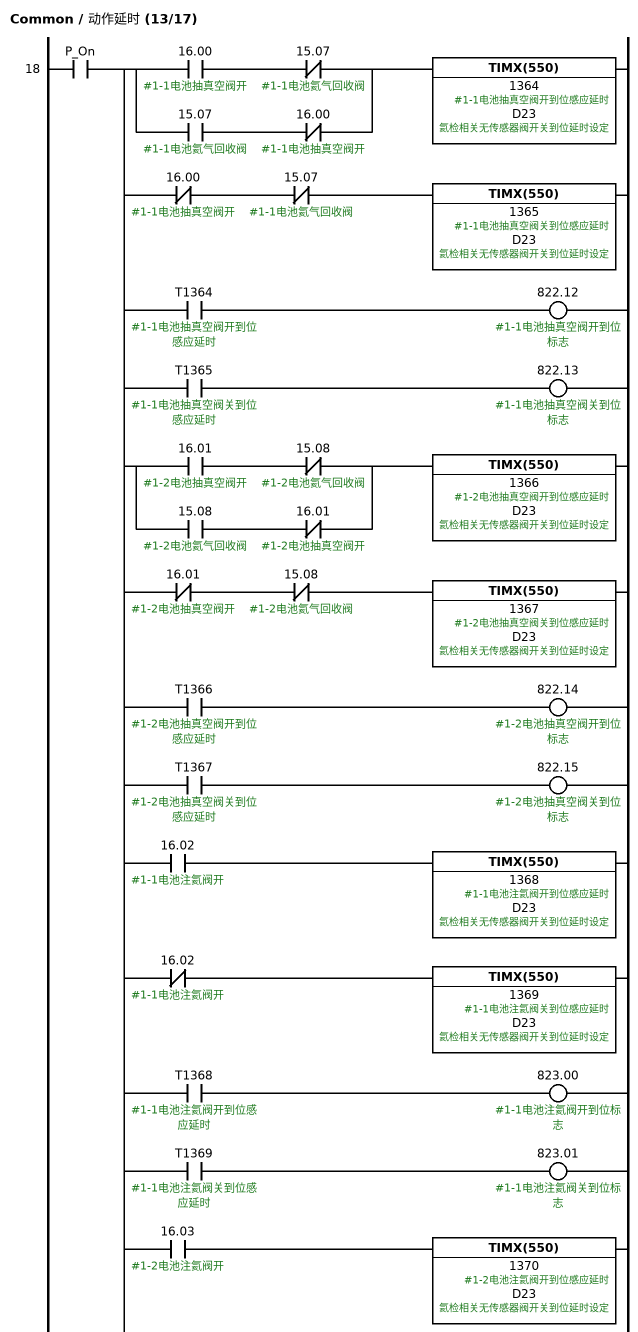

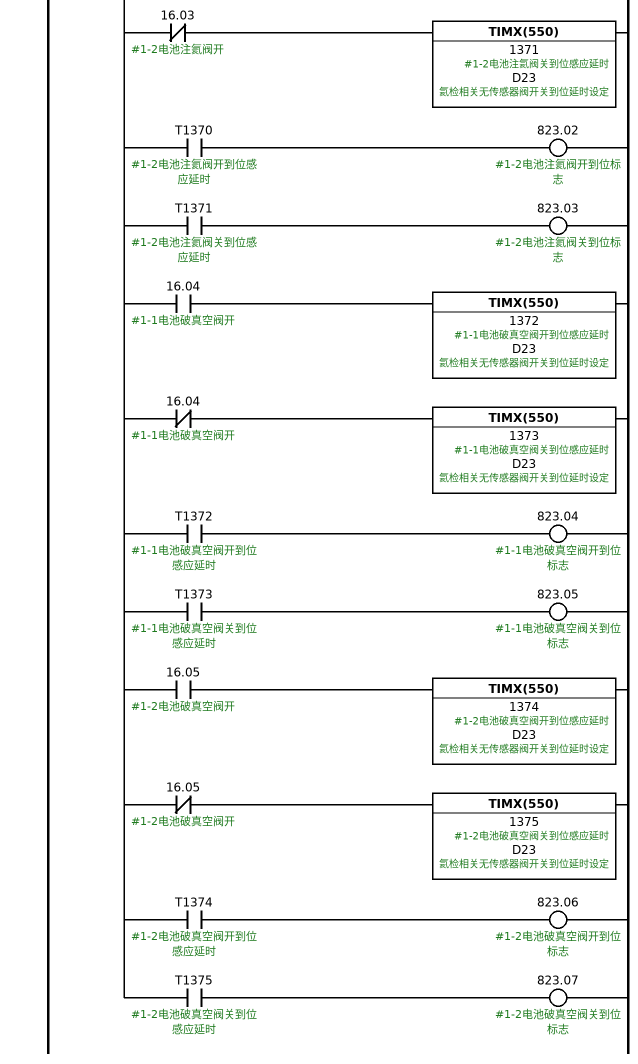
; rung 18
LD P_On
OUT TR0
LD 16.00  ; #1-1电池抽真空阀开
ANDNOT 15.07  ; #1-1电池氦气回收阀
LD 15.07  ; #1-1电池氦气回收阀
ANDNOT 16.00  ; #1-1电池抽真空阀开
ORLD
ANDLD
TIMX(550) 1364 D23  ; 氦检相关无传感器阀开关到位延时设定, #1-1电池抽真空阀开到位感应延时
LD TR0
ANDNOT 16.00  ; #1-1电池抽真空阀开
ANDNOT 15.07  ; #1-1电池氦气回收阀
TIMX(550) 1365 D23  ; 氦检相关无传感器阀开关到位延时设定, #1-1电池抽真空阀关到位感应延时
LD TR0
AND T1364  ; #1-1电池抽真空阀开到位感应延时
OUT 822.12  ; #1-1电池抽真空阀开到位标志
LD TR0
AND T1365  ; #1-1电池抽真空阀关到位感应延时
OUT 822.13  ; #1-1电池抽真空阀关到位标志
LD TR0
LD 16.01  ; #1-2电池抽真空阀开
ANDNOT 15.08  ; #1-2电池氦气回收阀
LD 15.08  ; #1-2电池氦气回收阀
ANDNOT 16.01  ; #1-2电池抽真空阀开
ORLD
ANDLD
TIMX(550) 1366 D23  ; 氦检相关无传感器阀开关到位延时设定, #1-2电池抽真空阀开到位感应延时
LD TR0
ANDNOT 16.01  ; #1-2电池抽真空阀开
ANDNOT 15.08  ; #1-2电池氦气回收阀
TIMX(550) 1367 D23  ; 氦检相关无传感器阀开关到位延时设定, #1-2电池抽真空阀关到位感应延时
LD TR0
AND T1366  ; #1-2电池抽真空阀开到位感应延时
OUT 822.14  ; #1-2电池抽真空阀开到位标志
LD TR0
AND T1367  ; #1-2电池抽真空阀关到位感应延时
OUT 822.15  ; #1-2电池抽真空阀关到位标志
LD TR0
AND 16.02  ; #1-1电池注氦阀开
TIMX(550) 1368 D23  ; 氦检相关无传感器阀开关到位延时设定, #1-1电池注氦阀开到位感应延时
LD TR0
ANDNOT 16.02  ; #1-1电池注氦阀开
TIMX(550) 1369 D23  ; 氦检相关无传感器阀开关到位延时设定, #1-1电池注氦阀关到位感应延时
LD TR0
AND T1368  ; #1-1电池注氦阀开到位感应延时
OUT 823.00  ; #1-1电池注氦阀开到位标志
LD TR0
AND T1369  ; #1-1电池注氦阀关到位感应延时
OUT 823.01  ; #1-1电池注氦阀关到位标志
LD TR0
AND 16.03  ; #1-2电池注氦阀开
TIMX(550) 1370 D23  ; 氦检相关无传感器阀开关到位延时设定, #1-2电池注氦阀开到位感应延时
LD TR0
ANDNOT 16.03  ; #1-2电池注氦阀开
TIMX(550) 1371 D23  ; 氦检相关无传感器阀开关到位延时设定, #1-2电池注氦阀关到位感应延时
LD TR0
AND T1370  ; #1-2电池注氦阀开到位感应延时
OUT 823.02  ; #1-2电池注氦阀开到位标志
LD TR0
AND T1371  ; #1-2电池注氦阀关到位感应延时
OUT 823.03  ; #1-2电池注氦阀关到位标志
LD TR0
AND 16.04  ; #1-1电池破真空阀开
TIMX(550) 1372 D23  ; 氦检相关无传感器阀开关到位延时设定, #1-1电池破真空阀开到位感应延时
LD TR0
ANDNOT 16.04  ; #1-1电池破真空阀开
TIMX(550) 1373 D23  ; 氦检相关无传感器阀开关到位延时设定, #1-1电池破真空阀关到位感应延时
LD TR0
AND T1372  ; #1-1电池破真空阀开到位感应延时
OUT 823.04  ; #1-1电池破真空阀开到位标志
LD TR0
AND T1373  ; #1-1电池破真空阀关到位感应延时
OUT 823.05  ; #1-1电池破真空阀关到位标志
LD TR0
AND 16.05  ; #1-2电池破真空阀开
TIMX(550) 1374 D23  ; 氦检相关无传感器阀开关到位延时设定, #1-2电池破真空阀开到位感应延时
LD TR0
ANDNOT 16.05  ; #1-2电池破真空阀开
TIMX(550) 1375 D23  ; 氦检相关无传感器阀开关到位延时设定, #1-2电池破真空阀关到位感应延时
LD TR0
AND T1374  ; #1-2电池破真空阀开到位感应延时
OUT 823.06  ; #1-2电池破真空阀开到位标志
LD TR0
AND T1375  ; #1-2电池破真空阀关到位感应延时
OUT 823.07  ; #1-2电池破真空阀关到位标志

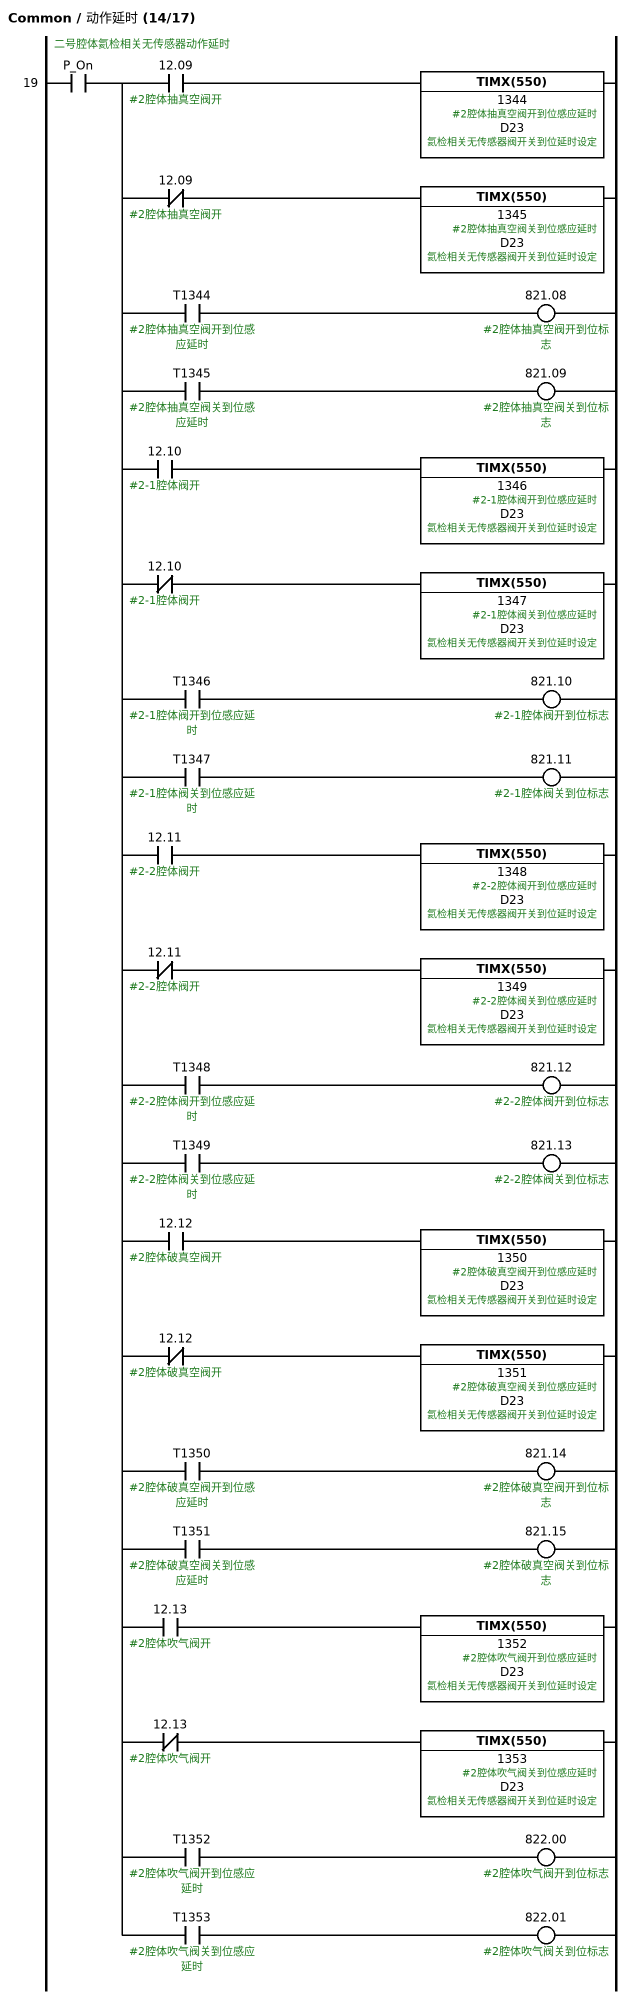
; rung 19: 二号腔体氦检相关无传感器动作延时
LD P_On
OUT TR0
AND 12.09  ; #2腔体抽真空阀开
TIMX(550) 1344 D23  ; 氦检相关无传感器阀开关到位延时设定, #2腔体抽真空阀开到位感应延时
LD TR0
ANDNOT 12.09  ; #2腔体抽真空阀开
TIMX(550) 1345 D23  ; 氦检相关无传感器阀开关到位延时设定, #2腔体抽真空阀关到位感应延时
LD TR0
AND T1344  ; #2腔体抽真空阀开到位感应延时
OUT 821.08  ; #2腔体抽真空阀开到位标志
LD TR0
AND T1345  ; #2腔体抽真空阀关到位感应延时
OUT 821.09  ; #2腔体抽真空阀关到位标志
LD TR0
AND 12.10  ; #2-1腔体阀开
TIMX(550) 1346 D23  ; 氦检相关无传感器阀开关到位延时设定, #2-1腔体阀开到位感应延时
LD TR0
ANDNOT 12.10  ; #2-1腔体阀开
TIMX(550) 1347 D23  ; 氦检相关无传感器阀开关到位延时设定, #2-1腔体阀关到位感应延时
LD TR0
AND T1346  ; #2-1腔体阀开到位感应延时
OUT 821.10  ; #2-1腔体阀开到位标志
LD TR0
AND T1347  ; #2-1腔体阀关到位感应延时
OUT 821.11  ; #2-1腔体阀关到位标志
LD TR0
AND 12.11  ; #2-2腔体阀开
TIMX(550) 1348 D23  ; 氦检相关无传感器阀开关到位延时设定, #2-2腔体阀开到位感应延时
LD TR0
ANDNOT 12.11  ; #2-2腔体阀开
TIMX(550) 1349 D23  ; 氦检相关无传感器阀开关到位延时设定, #2-2腔体阀关到位感应延时
LD TR0
AND T1348  ; #2-2腔体阀开到位感应延时
OUT 821.12  ; #2-2腔体阀开到位标志
LD TR0
AND T1349  ; #2-2腔体阀关到位感应延时
OUT 821.13  ; #2-2腔体阀关到位标志
LD TR0
AND 12.12  ; #2腔体破真空阀开
TIMX(550) 1350 D23  ; 氦检相关无传感器阀开关到位延时设定, #2腔体破真空阀开到位感应延时
LD TR0
ANDNOT 12.12  ; #2腔体破真空阀开
TIMX(550) 1351 D23  ; 氦检相关无传感器阀开关到位延时设定, #2腔体破真空阀关到位感应延时
LD TR0
AND T1350  ; #2腔体破真空阀开到位感应延时
OUT 821.14  ; #2腔体破真空阀开到位标志
LD TR0
AND T1351  ; #2腔体破真空阀关到位感应延时
OUT 821.15  ; #2腔体破真空阀关到位标志
LD TR0
AND 12.13  ; #2腔体吹气阀开
TIMX(550) 1352 D23  ; 氦检相关无传感器阀开关到位延时设定, #2腔体吹气阀开到位感应延时
LD TR0
ANDNOT 12.13  ; #2腔体吹气阀开
TIMX(550) 1353 D23  ; 氦检相关无传感器阀开关到位延时设定, #2腔体吹气阀关到位感应延时
LD TR0
AND T1352  ; #2腔体吹气阀开到位感应延时
OUT 822.00  ; #2腔体吹气阀开到位标志
LD TR0
AND T1353  ; #2腔体吹气阀关到位感应延时
OUT 822.01  ; #2腔体吹气阀关到位标志

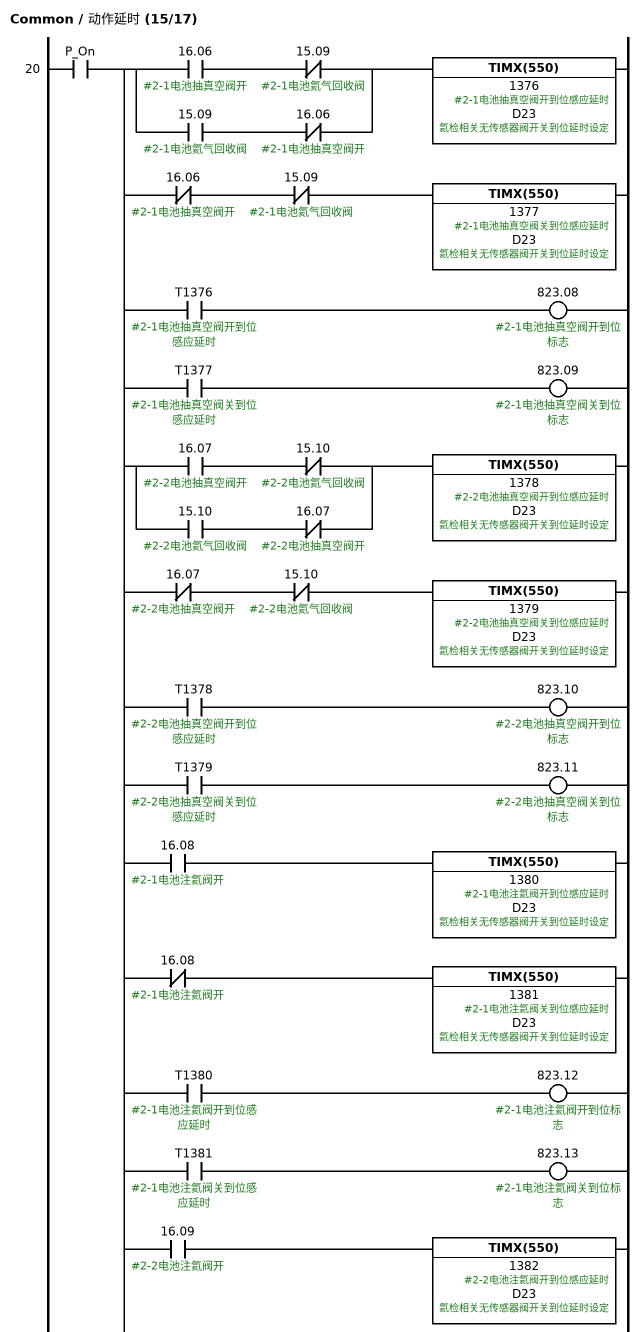

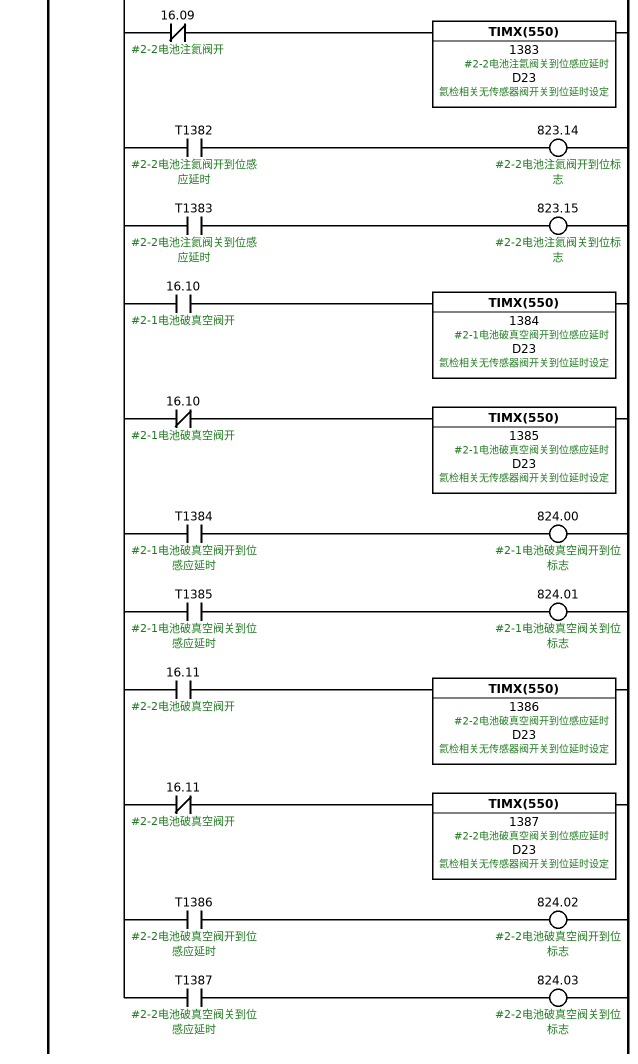
; rung 20
LD P_On
OUT TR0
LD 16.06  ; #2-1电池抽真空阀开
ANDNOT 15.09  ; #2-1电池氦气回收阀
LD 15.09  ; #2-1电池氦气回收阀
ANDNOT 16.06  ; #2-1电池抽真空阀开
ORLD
ANDLD
TIMX(550) 1376 D23  ; 氦检相关无传感器阀开关到位延时设定, #2-1电池抽真空阀开到位感应延时
LD TR0
ANDNOT 16.06  ; #2-1电池抽真空阀开
ANDNOT 15.09  ; #2-1电池氦气回收阀
TIMX(550) 1377 D23  ; 氦检相关无传感器阀开关到位延时设定, #2-1电池抽真空阀关到位感应延时
LD TR0
AND T1376  ; #2-1电池抽真空阀开到位感应延时
OUT 823.08  ; #2-1电池抽真空阀开到位标志
LD TR0
AND T1377  ; #2-1电池抽真空阀关到位感应延时
OUT 823.09  ; #2-1电池抽真空阀关到位标志
LD TR0
LD 16.07  ; #2-2电池抽真空阀开
ANDNOT 15.10  ; #2-2电池氦气回收阀
LD 15.10  ; #2-2电池氦气回收阀
ANDNOT 16.07  ; #2-2电池抽真空阀开
ORLD
ANDLD
TIMX(550) 1378 D23  ; 氦检相关无传感器阀开关到位延时设定, #2-2电池抽真空阀开到位感应延时
LD TR0
ANDNOT 16.07  ; #2-2电池抽真空阀开
ANDNOT 15.10  ; #2-2电池氦气回收阀
TIMX(550) 1379 D23  ; 氦检相关无传感器阀开关到位延时设定, #2-2电池抽真空阀关到位感应延时
LD TR0
AND T1378  ; #2-2电池抽真空阀开到位感应延时
OUT 823.10  ; #2-2电池抽真空阀开到位标志
LD TR0
AND T1379  ; #2-2电池抽真空阀关到位感应延时
OUT 823.11  ; #2-2电池抽真空阀关到位标志
LD TR0
AND 16.08  ; #2-1电池注氦阀开
TIMX(550) 1380 D23  ; 氦检相关无传感器阀开关到位延时设定, #2-1电池注氦阀开到位感应延时
LD TR0
ANDNOT 16.08  ; #2-1电池注氦阀开
TIMX(550) 1381 D23  ; 氦检相关无传感器阀开关到位延时设定, #2-1电池注氦阀关到位感应延时
LD TR0
AND T1380  ; #2-1电池注氦阀开到位感应延时
OUT 823.12  ; #2-1电池注氦阀开到位标志
LD TR0
AND T1381  ; #2-1电池注氦阀关到位感应延时
OUT 823.13  ; #2-1电池注氦阀关到位标志
LD TR0
AND 16.09  ; #2-2电池注氦阀开
TIMX(550) 1382 D23  ; 氦检相关无传感器阀开关到位延时设定, #2-2电池注氦阀开到位感应延时
LD TR0
ANDNOT 16.09  ; #2-2电池注氦阀开
TIMX(550) 1383 D23  ; 氦检相关无传感器阀开关到位延时设定, #2-2电池注氦阀关到位感应延时
LD TR0
AND T1382  ; #2-2电池注氦阀开到位感应延时
OUT 823.14  ; #2-2电池注氦阀开到位标志
LD TR0
AND T1383  ; #2-2电池注氦阀关到位感应延时
OUT 823.15  ; #2-2电池注氦阀关到位标志
LD TR0
AND 16.10  ; #2-1电池破真空阀开
TIMX(550) 1384 D23  ; 氦检相关无传感器阀开关到位延时设定, #2-1电池破真空阀开到位感应延时
LD TR0
ANDNOT 16.10  ; #2-1电池破真空阀开
TIMX(550) 1385 D23  ; 氦检相关无传感器阀开关到位延时设定, #2-1电池破真空阀关到位感应延时
LD TR0
AND T1384  ; #2-1电池破真空阀开到位感应延时
OUT 824.00  ; #2-1电池破真空阀开到位标志
LD TR0
AND T1385  ; #2-1电池破真空阀关到位感应延时
OUT 824.01  ; #2-1电池破真空阀关到位标志
LD TR0
AND 16.11  ; #2-2电池破真空阀开
TIMX(550) 1386 D23  ; 氦检相关无传感器阀开关到位延时设定, #2-2电池破真空阀开到位感应延时
LD TR0
ANDNOT 16.11  ; #2-2电池破真空阀开
TIMX(550) 1387 D23  ; 氦检相关无传感器阀开关到位延时设定, #2-2电池破真空阀关到位感应延时
LD TR0
AND T1386  ; #2-2电池破真空阀开到位感应延时
OUT 824.02  ; #2-2电池破真空阀开到位标志
LD TR0
AND T1387  ; #2-2电池破真空阀关到位感应延时
OUT 824.03  ; #2-2电池破真空阀关到位标志

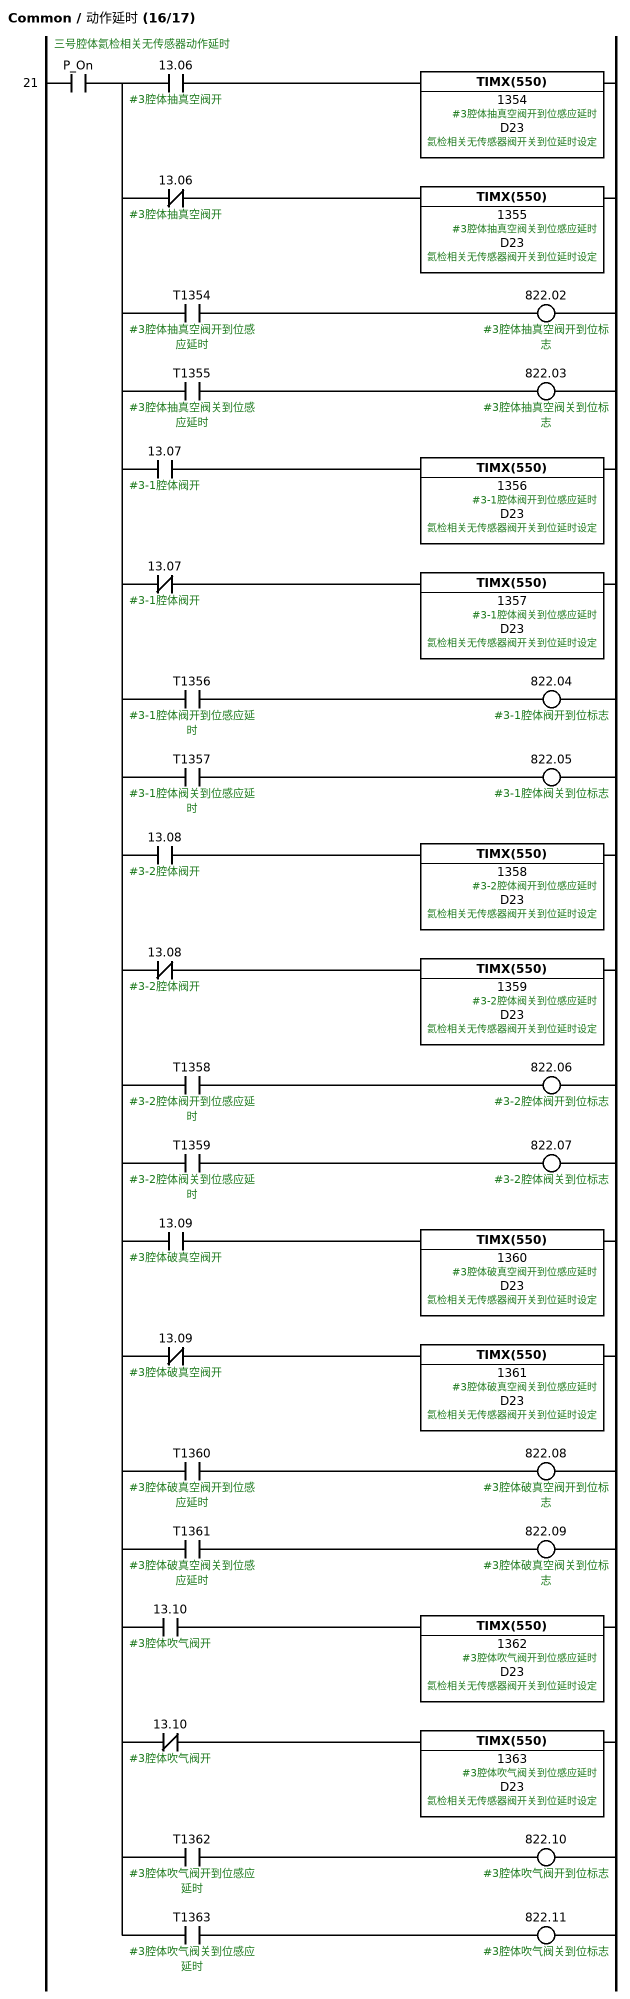
; rung 21: 三号腔体氦检相关无传感器动作延时
LD P_On
OUT TR0
AND 13.06  ; #3腔体抽真空阀开
TIMX(550) 1354 D23  ; 氦检相关无传感器阀开关到位延时设定, #3腔体抽真空阀开到位感应延时
LD TR0
ANDNOT 13.06  ; #3腔体抽真空阀开
TIMX(550) 1355 D23  ; 氦检相关无传感器阀开关到位延时设定, #3腔体抽真空阀关到位感应延时
LD TR0
AND T1354  ; #3腔体抽真空阀开到位感应延时
OUT 822.02  ; #3腔体抽真空阀开到位标志
LD TR0
AND T1355  ; #3腔体抽真空阀关到位感应延时
OUT 822.03  ; #3腔体抽真空阀关到位标志
LD TR0
AND 13.07  ; #3-1腔体阀开
TIMX(550) 1356 D23  ; 氦检相关无传感器阀开关到位延时设定, #3-1腔体阀开到位感应延时
LD TR0
ANDNOT 13.07  ; #3-1腔体阀开
TIMX(550) 1357 D23  ; 氦检相关无传感器阀开关到位延时设定, #3-1腔体阀关到位感应延时
LD TR0
AND T1356  ; #3-1腔体阀开到位感应延时
OUT 822.04  ; #3-1腔体阀开到位标志
LD TR0
AND T1357  ; #3-1腔体阀关到位感应延时
OUT 822.05  ; #3-1腔体阀关到位标志
LD TR0
AND 13.08  ; #3-2腔体阀开
TIMX(550) 1358 D23  ; 氦检相关无传感器阀开关到位延时设定, #3-2腔体阀开到位感应延时
LD TR0
ANDNOT 13.08  ; #3-2腔体阀开
TIMX(550) 1359 D23  ; 氦检相关无传感器阀开关到位延时设定, #3-2腔体阀关到位感应延时
LD TR0
AND T1358  ; #3-2腔体阀开到位感应延时
OUT 822.06  ; #3-2腔体阀开到位标志
LD TR0
AND T1359  ; #3-2腔体阀关到位感应延时
OUT 822.07  ; #3-2腔体阀关到位标志
LD TR0
AND 13.09  ; #3腔体破真空阀开
TIMX(550) 1360 D23  ; 氦检相关无传感器阀开关到位延时设定, #3腔体破真空阀开到位感应延时
LD TR0
ANDNOT 13.09  ; #3腔体破真空阀开
TIMX(550) 1361 D23  ; 氦检相关无传感器阀开关到位延时设定, #3腔体破真空阀关到位感应延时
LD TR0
AND T1360  ; #3腔体破真空阀开到位感应延时
OUT 822.08  ; #3腔体破真空阀开到位标志
LD TR0
AND T1361  ; #3腔体破真空阀关到位感应延时
OUT 822.09  ; #3腔体破真空阀关到位标志
LD TR0
AND 13.10  ; #3腔体吹气阀开
TIMX(550) 1362 D23  ; 氦检相关无传感器阀开关到位延时设定, #3腔体吹气阀开到位感应延时
LD TR0
ANDNOT 13.10  ; #3腔体吹气阀开
TIMX(550) 1363 D23  ; 氦检相关无传感器阀开关到位延时设定, #3腔体吹气阀关到位感应延时
LD TR0
AND T1362  ; #3腔体吹气阀开到位感应延时
OUT 822.10  ; #3腔体吹气阀开到位标志
LD TR0
AND T1363  ; #3腔体吹气阀关到位感应延时
OUT 822.11  ; #3腔体吹气阀关到位标志

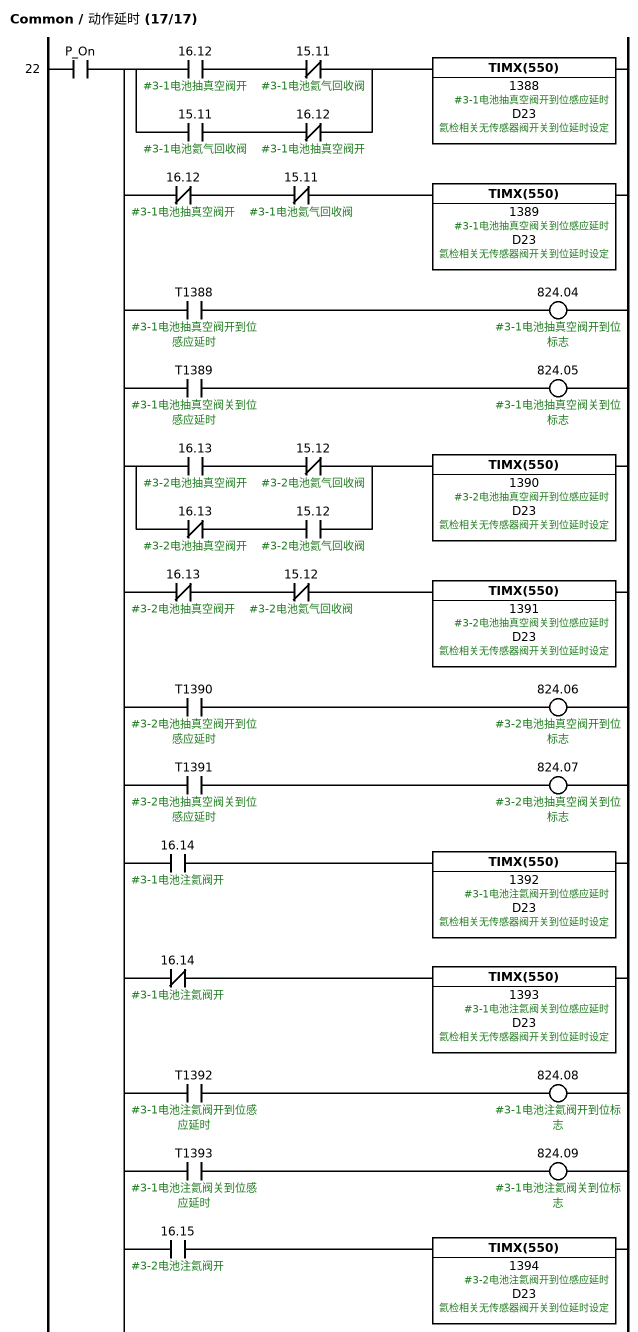

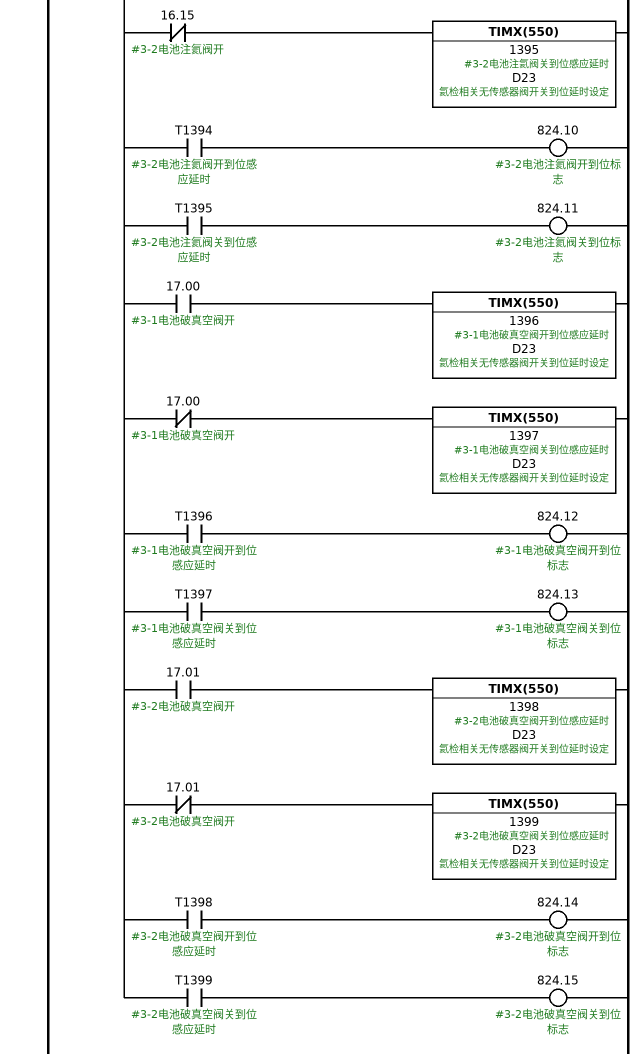
; rung 22
LD P_On
OUT TR0
LD 16.12  ; #3-1电池抽真空阀开
ANDNOT 15.11  ; #3-1电池氦气回收阀
LD 15.11  ; #3-1电池氦气回收阀
ANDNOT 16.12  ; #3-1电池抽真空阀开
ORLD
ANDLD
TIMX(550) 1388 D23  ; 氦检相关无传感器阀开关到位延时设定, #3-1电池抽真空阀开到位感应延时
LD TR0
ANDNOT 16.12  ; #3-1电池抽真空阀开
ANDNOT 15.11  ; #3-1电池氦气回收阀
TIMX(550) 1389 D23  ; 氦检相关无传感器阀开关到位延时设定, #3-1电池抽真空阀关到位感应延时
LD TR0
AND T1388  ; #3-1电池抽真空阀开到位感应延时
OUT 824.04  ; #3-1电池抽真空阀开到位标志
LD TR0
AND T1389  ; #3-1电池抽真空阀关到位感应延时
OUT 824.05  ; #3-1电池抽真空阀关到位标志
LD TR0
LD 16.13  ; #3-2电池抽真空阀开
ANDNOT 15.12  ; #3-2电池氦气回收阀
LDNOT 16.13  ; #3-2电池抽真空阀开
AND 15.12  ; #3-2电池氦气回收阀
ORLD
ANDLD
TIMX(550) 1390 D23  ; 氦检相关无传感器阀开关到位延时设定, #3-2电池抽真空阀开到位感应延时
LD TR0
ANDNOT 16.13  ; #3-2电池抽真空阀开
ANDNOT 15.12  ; #3-2电池氦气回收阀
TIMX(550) 1391 D23  ; 氦检相关无传感器阀开关到位延时设定, #3-2电池抽真空阀关到位感应延时
LD TR0
AND T1390  ; #3-2电池抽真空阀开到位感应延时
OUT 824.06  ; #3-2电池抽真空阀开到位标志
LD TR0
AND T1391  ; #3-2电池抽真空阀关到位感应延时
OUT 824.07  ; #3-2电池抽真空阀关到位标志
LD TR0
AND 16.14  ; #3-1电池注氦阀开
TIMX(550) 1392 D23  ; 氦检相关无传感器阀开关到位延时设定, #3-1电池注氦阀开到位感应延时
LD TR0
ANDNOT 16.14  ; #3-1电池注氦阀开
TIMX(550) 1393 D23  ; 氦检相关无传感器阀开关到位延时设定, #3-1电池注氦阀关到位感应延时
LD TR0
AND T1392  ; #3-1电池注氦阀开到位感应延时
OUT 824.08  ; #3-1电池注氦阀开到位标志
LD TR0
AND T1393  ; #3-1电池注氦阀关到位感应延时
OUT 824.09  ; #3-1电池注氦阀关到位标志
LD TR0
AND 16.15  ; #3-2电池注氦阀开
TIMX(550) 1394 D23  ; 氦检相关无传感器阀开关到位延时设定, #3-2电池注氦阀开到位感应延时
LD TR0
ANDNOT 16.15  ; #3-2电池注氦阀开
TIMX(550) 1395 D23  ; 氦检相关无传感器阀开关到位延时设定, #3-2电池注氦阀关到位感应延时
LD TR0
AND T1394  ; #3-2电池注氦阀开到位感应延时
OUT 824.10  ; #3-2电池注氦阀开到位标志
LD TR0
AND T1395  ; #3-2电池注氦阀关到位感应延时
OUT 824.11  ; #3-2电池注氦阀关到位标志
LD TR0
AND 17.00  ; #3-1电池破真空阀开
TIMX(550) 1396 D23  ; 氦检相关无传感器阀开关到位延时设定, #3-1电池破真空阀开到位感应延时
LD TR0
ANDNOT 17.00  ; #3-1电池破真空阀开
TIMX(550) 1397 D23  ; 氦检相关无传感器阀开关到位延时设定, #3-1电池破真空阀关到位感应延时
LD TR0
AND T1396  ; #3-1电池破真空阀开到位感应延时
OUT 824.12  ; #3-1电池破真空阀开到位标志
LD TR0
AND T1397  ; #3-1电池破真空阀关到位感应延时
OUT 824.13  ; #3-1电池破真空阀关到位标志
LD TR0
AND 17.01  ; #3-2电池破真空阀开
TIMX(550) 1398 D23  ; 氦检相关无传感器阀开关到位延时设定, #3-2电池破真空阀开到位感应延时
LD TR0
ANDNOT 17.01  ; #3-2电池破真空阀开
TIMX(550) 1399 D23  ; 氦检相关无传感器阀开关到位延时设定, #3-2电池破真空阀关到位感应延时
LD TR0
AND T1398  ; #3-2电池破真空阀开到位感应延时
OUT 824.14  ; #3-2电池破真空阀开到位标志
LD TR0
AND T1399  ; #3-2电池破真空阀关到位感应延时
OUT 824.15  ; #3-2电池破真空阀关到位标志

### Section 传感器延时

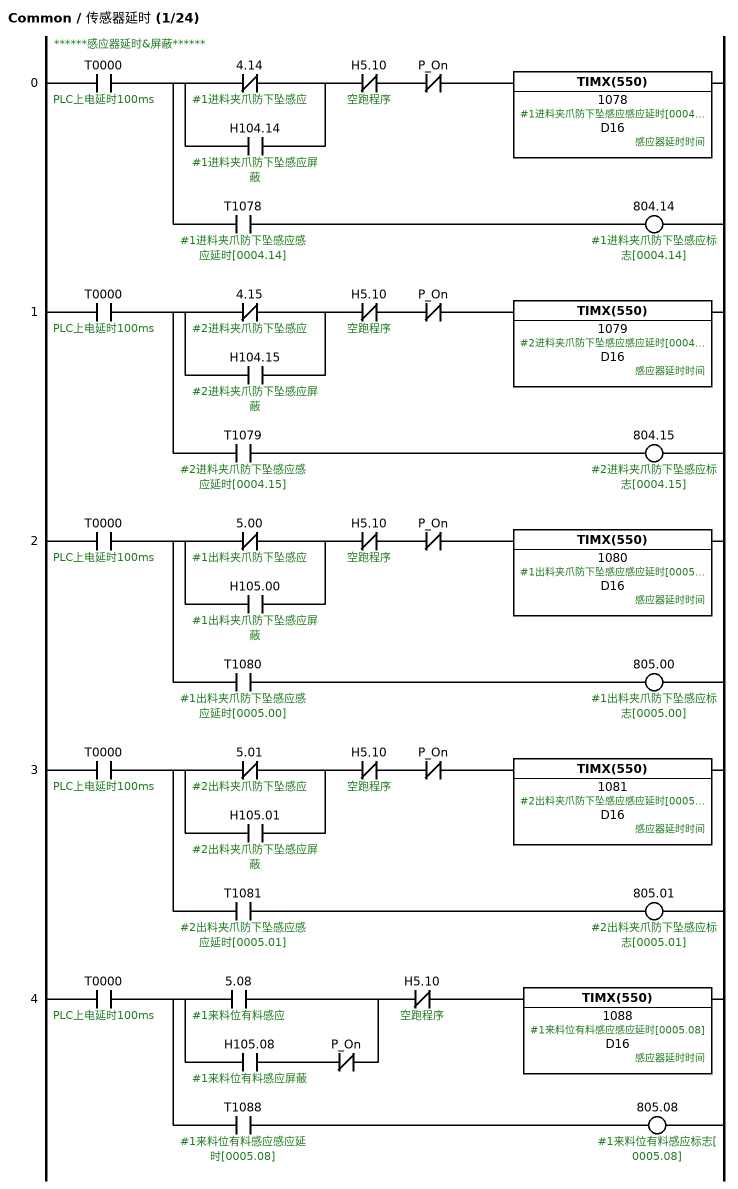
; rung 0: ******感应器延时&屏蔽******
LD T0000  ; PLC上电延时100ms
OUT TR0
LDNOT 4.14  ; #1进料夹爪防下坠感应
OR H104.14  ; #1进料夹爪防下坠感应屏蔽
ANDLD
ANDNOT H5.10  ; 空跑程序
ANDNOT P_On
TIMX(550) 1078 D16  ; 感应器延时时间, #1进料夹爪防下坠感应感应延时[0004.14]
LD TR0
AND T1078  ; #1进料夹爪防下坠感应感应延时[0004.14]
OUT 804.14  ; #1进料夹爪防下坠感应标志[0004.14]
; rung 1
LD T0000  ; PLC上电延时100ms
OUT TR0
LDNOT 4.15  ; #2进料夹爪防下坠感应
OR H104.15  ; #2进料夹爪防下坠感应屏蔽
ANDLD
ANDNOT H5.10  ; 空跑程序
ANDNOT P_On
TIMX(550) 1079 D16  ; 感应器延时时间, #2进料夹爪防下坠感应感应延时[0004.15]
LD TR0
AND T1079  ; #2进料夹爪防下坠感应感应延时[0004.15]
OUT 804.15  ; #2进料夹爪防下坠感应标志[0004.15]
; rung 2
LD T0000  ; PLC上电延时100ms
OUT TR0
LDNOT 5.00  ; #1出料夹爪防下坠感应
OR H105.00  ; #1出料夹爪防下坠感应屏蔽
ANDLD
ANDNOT H5.10  ; 空跑程序
ANDNOT P_On
TIMX(550) 1080 D16  ; 感应器延时时间, #1出料夹爪防下坠感应感应延时[0005.00]
LD TR0
AND T1080  ; #1出料夹爪防下坠感应感应延时[0005.00]
OUT 805.00  ; #1出料夹爪防下坠感应标志[0005.00]
; rung 3
LD T0000  ; PLC上电延时100ms
OUT TR0
LDNOT 5.01  ; #2出料夹爪防下坠感应
OR H105.01  ; #2出料夹爪防下坠感应屏蔽
ANDLD
ANDNOT H5.10  ; 空跑程序
ANDNOT P_On
TIMX(550) 1081 D16  ; 感应器延时时间, #2出料夹爪防下坠感应感应延时[0005.01]
LD TR0
AND T1081  ; #2出料夹爪防下坠感应感应延时[0005.01]
OUT 805.01  ; #2出料夹爪防下坠感应标志[0005.01]
; rung 4
LD T0000  ; PLC上电延时100ms
OUT TR0
LD 5.08  ; #1来料位有料感应
LD H105.08  ; #1来料位有料感应屏蔽
ANDNOT P_On
ORLD
ANDLD
ANDNOT H5.10  ; 空跑程序
TIMX(550) 1088 D16  ; 感应器延时时间, #1来料位有料感应感应延时[0005.08]
LD TR0
AND T1088  ; #1来料位有料感应感应延时[0005.08]
OUT 805.08  ; #1来料位有料感应标志[0005.08]

